REGION Network 1
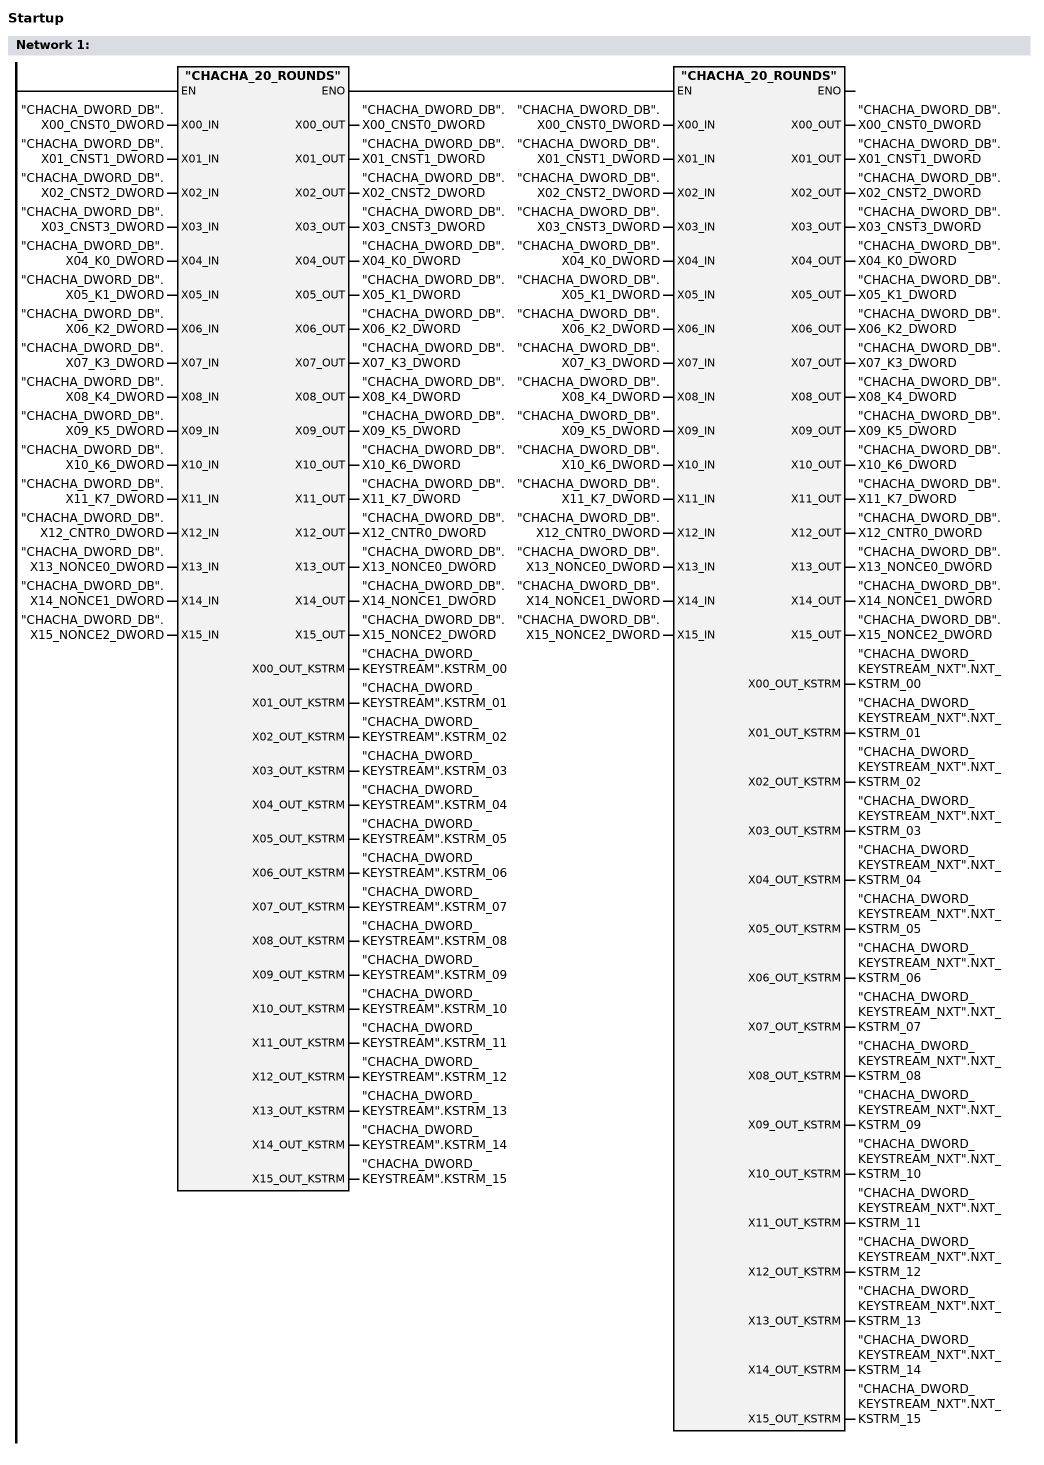
   RUNG wire#powerrail
      "CHACHA_20_ROUNDS"(X00_IN := "CHACHA_DWORD_DB".X00_CNST0_DWORD, X01_IN := "CHACHA_DWORD_DB".X01_CNST1_DWORD, X02_IN := "CHACHA_DWORD_DB".X02_CNST2_DWORD, X03_IN := "CHACHA_DWORD_DB".X03_CNST3_DWORD, X04_IN := "CHACHA_DWORD_DB".X04_K0_DWORD, X05_IN := "CHACHA_DWORD_DB".X05_K1_DWORD, X06_IN := "CHACHA_DWORD_DB".X06_K2_DWORD, X07_IN := "CHACHA_DWORD_DB".X07_K3_DWORD, X08_IN := "CHACHA_DWORD_DB".X08_K4_DWORD, X09_IN := "CHACHA_DWORD_DB".X09_K5_DWORD, X10_IN := "CHACHA_DWORD_DB".X10_K6_DWORD, X11_IN := "CHACHA_DWORD_DB".X11_K7_DWORD, X12_IN := "CHACHA_DWORD_DB".X12_CNTR0_DWORD, X13_IN := "CHACHA_DWORD_DB".X13_NONCE0_DWORD, X14_IN := "CHACHA_DWORD_DB".X14_NONCE1_DWORD, X15_IN := "CHACHA_DWORD_DB".X15_NONCE2_DWORD, X00_OUT => "CHACHA_DWORD_DB".X00_CNST0_DWORD, X01_OUT => "CHACHA_DWORD_DB".X01_CNST1_DWORD, X02_OUT => "CHACHA_DWORD_DB".X02_CNST2_DWORD, X03_OUT => "CHACHA_DWORD_DB".X03_CNST3_DWORD, X04_OUT => "CHACHA_DWORD_DB".X04_K0_DWORD, X05_OUT => "CHACHA_DWORD_DB".X05_K1_DWORD, X06_OUT => "CHACHA_DWORD_DB".X06_K2_DWORD, X07_OUT => "CHACHA_DWORD_DB".X07_K3_DWORD, X08_OUT => "CHACHA_DWORD_DB".X08_K4_DWORD, X09_OUT => "CHACHA_DWORD_DB".X09_K5_DWORD, X10_OUT => "CHACHA_DWORD_DB".X10_K6_DWORD, X11_OUT => "CHACHA_DWORD_DB".X11_K7_DWORD, X12_OUT => "CHACHA_DWORD_DB".X12_CNTR0_DWORD, X13_OUT => "CHACHA_DWORD_DB".X13_NONCE0_DWORD, X14_OUT => "CHACHA_DWORD_DB".X14_NONCE1_DWORD, X15_OUT => "CHACHA_DWORD_DB".X15_NONCE2_DWORD, X00_OUT_KSTRM => "CHACHA_DWORD_KEYSTREAM".KSTRM_00, X01_OUT_KSTRM => "CHACHA_DWORD_KEYSTREAM".KSTRM_01, X02_OUT_KSTRM => "CHACHA_DWORD_KEYSTREAM".KSTRM_02, X03_OUT_KSTRM => "CHACHA_DWORD_KEYSTREAM".KSTRM_03, X04_OUT_KSTRM => "CHACHA_DWORD_KEYSTREAM".KSTRM_04, X05_OUT_KSTRM => "CHACHA_DWORD_KEYSTREAM".KSTRM_05, X06_OUT_KSTRM => "CHACHA_DWORD_KEYSTREAM".KSTRM_06, X07_OUT_KSTRM => "CHACHA_DWORD_KEYSTREAM".KSTRM_07, X08_OUT_KSTRM => "CHACHA_DWORD_KEYSTREAM".KSTRM_08, X09_OUT_KSTRM => "CHACHA_DWORD_KEYSTREAM".KSTRM_09, X10_OUT_KSTRM => "CHACHA_DWORD_KEYSTREAM".KSTRM_10, X11_OUT_KSTRM => "CHACHA_DWORD_KEYSTREAM".KSTRM_11, X12_OUT_KSTRM => "CHACHA_DWORD_KEYSTREAM".KSTRM_12, X13_OUT_KSTRM => "CHACHA_DWORD_KEYSTREAM".KSTRM_13, X14_OUT_KSTRM => "CHACHA_DWORD_KEYSTREAM".KSTRM_14, X15_OUT_KSTRM => "CHACHA_DWORD_KEYSTREAM".KSTRM_15)
      "CHACHA_20_ROUNDS"(X00_IN := "CHACHA_DWORD_DB".X00_CNST0_DWORD, X01_IN := "CHACHA_DWORD_DB".X01_CNST1_DWORD, X02_IN := "CHACHA_DWORD_DB".X02_CNST2_DWORD, X03_IN := "CHACHA_DWORD_DB".X03_CNST3_DWORD, X04_IN := "CHACHA_DWORD_DB".X04_K0_DWORD, X05_IN := "CHACHA_DWORD_DB".X05_K1_DWORD, X06_IN := "CHACHA_DWORD_DB".X06_K2_DWORD, X07_IN := "CHACHA_DWORD_DB".X07_K3_DWORD, X08_IN := "CHACHA_DWORD_DB".X08_K4_DWORD, X09_IN := "CHACHA_DWORD_DB".X09_K5_DWORD, X10_IN := "CHACHA_DWORD_DB".X10_K6_DWORD, X11_IN := "CHACHA_DWORD_DB".X11_K7_DWORD, X12_IN := "CHACHA_DWORD_DB".X12_CNTR0_DWORD, X13_IN := "CHACHA_DWORD_DB".X13_NONCE0_DWORD, X14_IN := "CHACHA_DWORD_DB".X14_NONCE1_DWORD, X15_IN := "CHACHA_DWORD_DB".X15_NONCE2_DWORD, X00_OUT => "CHACHA_DWORD_DB".X00_CNST0_DWORD, X01_OUT => "CHACHA_DWORD_DB".X01_CNST1_DWORD, X02_OUT => "CHACHA_DWORD_DB".X02_CNST2_DWORD, X03_OUT => "CHACHA_DWORD_DB".X03_CNST3_DWORD, X04_OUT => "CHACHA_DWORD_DB".X04_K0_DWORD, X05_OUT => "CHACHA_DWORD_DB".X05_K1_DWORD, X06_OUT => "CHACHA_DWORD_DB".X06_K2_DWORD, X07_OUT => "CHACHA_DWORD_DB".X07_K3_DWORD, X08_OUT => "CHACHA_DWORD_DB".X08_K4_DWORD, X09_OUT => "CHACHA_DWORD_DB".X09_K5_DWORD, X10_OUT => "CHACHA_DWORD_DB".X10_K6_DWORD, X11_OUT => "CHACHA_DWORD_DB".X11_K7_DWORD, X12_OUT => "CHACHA_DWORD_DB".X12_CNTR0_DWORD, X13_OUT => "CHACHA_DWORD_DB".X13_NONCE0_DWORD, X14_OUT => "CHACHA_DWORD_DB".X14_NONCE1_DWORD, X15_OUT => "CHACHA_DWORD_DB".X15_NONCE2_DWORD, X00_OUT_KSTRM => "CHACHA_DWORD_KEYSTREAM_NXT".NXT_KSTRM_00, X01_OUT_KSTRM => "CHACHA_DWORD_KEYSTREAM_NXT".NXT_KSTRM_01, X02_OUT_KSTRM => "CHACHA_DWORD_KEYSTREAM_NXT".NXT_KSTRM_02, X03_OUT_KSTRM => "CHACHA_DWORD_KEYSTREAM_NXT".NXT_KSTRM_03, X04_OUT_KSTRM => "CHACHA_DWORD_KEYSTREAM_NXT".NXT_KSTRM_04, X05_OUT_KSTRM => "CHACHA_DWORD_KEYSTREAM_NXT".NXT_KSTRM_05, X06_OUT_KSTRM => "CHACHA_DWORD_KEYSTREAM_NXT".NXT_KSTRM_06, X07_OUT_KSTRM => "CHACHA_DWORD_KEYSTREAM_NXT".NXT_KSTRM_07, X08_OUT_KSTRM => "CHACHA_DWORD_KEYSTREAM_NXT".NXT_KSTRM_08, X09_OUT_KSTRM => "CHACHA_DWORD_KEYSTREAM_NXT".NXT_KSTRM_09, X10_OUT_KSTRM => "CHACHA_DWORD_KEYSTREAM_NXT".NXT_KSTRM_10, X11_OUT_KSTRM => "CHACHA_DWORD_KEYSTREAM_NXT".NXT_KSTRM_11, X12_OUT_KSTRM => "CHACHA_DWORD_KEYSTREAM_NXT".NXT_KSTRM_12, X13_OUT_KSTRM => "CHACHA_DWORD_KEYSTREAM_NXT".NXT_KSTRM_13, X14_OUT_KSTRM => "CHACHA_DWORD_KEYSTREAM_NXT".NXT_KSTRM_14, X15_OUT_KSTRM => "CHACHA_DWORD_KEYSTREAM_NXT".NXT_KSTRM_15)
   END_RUNG
   // the same network as SCL:
   "CHACHA_20_ROUNDS"(X00_IN := "CHACHA_DWORD_DB".X00_CNST0_DWORD,
                      X01_IN := "CHACHA_DWORD_DB".X01_CNST1_DWORD,
                      X02_IN := "CHACHA_DWORD_DB".X02_CNST2_DWORD,
                      X03_IN := "CHACHA_DWORD_DB".X03_CNST3_DWORD,
                      X04_IN := "CHACHA_DWORD_DB".X04_K0_DWORD,
                      X05_IN := "CHACHA_DWORD_DB".X05_K1_DWORD,
                      X06_IN := "CHACHA_DWORD_DB".X06_K2_DWORD,
                      X07_IN := "CHACHA_DWORD_DB".X07_K3_DWORD,
                      X08_IN := "CHACHA_DWORD_DB".X08_K4_DWORD,
                      X09_IN := "CHACHA_DWORD_DB".X09_K5_DWORD,
                      X10_IN := "CHACHA_DWORD_DB".X10_K6_DWORD,
                      X11_IN := "CHACHA_DWORD_DB".X11_K7_DWORD,
                      X12_IN := "CHACHA_DWORD_DB".X12_CNTR0_DWORD,
                      X13_IN := "CHACHA_DWORD_DB".X13_NONCE0_DWORD,
                      X14_IN := "CHACHA_DWORD_DB".X14_NONCE1_DWORD,
                      X15_IN := "CHACHA_DWORD_DB".X15_NONCE2_DWORD,
                      X00_OUT => "CHACHA_DWORD_DB".X00_CNST0_DWORD,
                      X01_OUT => "CHACHA_DWORD_DB".X01_CNST1_DWORD,
                      X02_OUT => "CHACHA_DWORD_DB".X02_CNST2_DWORD,
                      X03_OUT => "CHACHA_DWORD_DB".X03_CNST3_DWORD,
                      X04_OUT => "CHACHA_DWORD_DB".X04_K0_DWORD,
                      X05_OUT => "CHACHA_DWORD_DB".X05_K1_DWORD,
                      X06_OUT => "CHACHA_DWORD_DB".X06_K2_DWORD,
                      X07_OUT => "CHACHA_DWORD_DB".X07_K3_DWORD,
                      X08_OUT => "CHACHA_DWORD_DB".X08_K4_DWORD,
                      X09_OUT => "CHACHA_DWORD_DB".X09_K5_DWORD,
                      X10_OUT => "CHACHA_DWORD_DB".X10_K6_DWORD,
                      X11_OUT => "CHACHA_DWORD_DB".X11_K7_DWORD,
                      X12_OUT => "CHACHA_DWORD_DB".X12_CNTR0_DWORD,
                      X13_OUT => "CHACHA_DWORD_DB".X13_NONCE0_DWORD,
                      X14_OUT => "CHACHA_DWORD_DB".X14_NONCE1_DWORD,
                      X15_OUT => "CHACHA_DWORD_DB".X15_NONCE2_DWORD,
                      X00_OUT_KSTRM => "CHACHA_DWORD_KEYSTREAM".KSTRM_00,
                      X01_OUT_KSTRM => "CHACHA_DWORD_KEYSTREAM".KSTRM_01,
                      X02_OUT_KSTRM => "CHACHA_DWORD_KEYSTREAM".KSTRM_02,
                      X03_OUT_KSTRM => "CHACHA_DWORD_KEYSTREAM".KSTRM_03,
                      X04_OUT_KSTRM => "CHACHA_DWORD_KEYSTREAM".KSTRM_04,
                      X05_OUT_KSTRM => "CHACHA_DWORD_KEYSTREAM".KSTRM_05,
                      X06_OUT_KSTRM => "CHACHA_DWORD_KEYSTREAM".KSTRM_06,
                      X07_OUT_KSTRM => "CHACHA_DWORD_KEYSTREAM".KSTRM_07,
                      X08_OUT_KSTRM => "CHACHA_DWORD_KEYSTREAM".KSTRM_08,
                      X09_OUT_KSTRM => "CHACHA_DWORD_KEYSTREAM".KSTRM_09,
                      X10_OUT_KSTRM => "CHACHA_DWORD_KEYSTREAM".KSTRM_10,
                      X11_OUT_KSTRM => "CHACHA_DWORD_KEYSTREAM".KSTRM_11,
                      X12_OUT_KSTRM => "CHACHA_DWORD_KEYSTREAM".KSTRM_12,
                      X13_OUT_KSTRM => "CHACHA_DWORD_KEYSTREAM".KSTRM_13,
                      X14_OUT_KSTRM => "CHACHA_DWORD_KEYSTREAM".KSTRM_14,
                      X15_OUT_KSTRM => "CHACHA_DWORD_KEYSTREAM".KSTRM_15,
                      ENO => #_w1);
   IF #_w1 THEN
       "CHACHA_20_ROUNDS"(X00_IN := "CHACHA_DWORD_DB".X00_CNST0_DWORD,
                          X01_IN := "CHACHA_DWORD_DB".X01_CNST1_DWORD,
                          X02_IN := "CHACHA_DWORD_DB".X02_CNST2_DWORD,
                          X03_IN := "CHACHA_DWORD_DB".X03_CNST3_DWORD,
                          X04_IN := "CHACHA_DWORD_DB".X04_K0_DWORD,
                          X05_IN := "CHACHA_DWORD_DB".X05_K1_DWORD,
                          X06_IN := "CHACHA_DWORD_DB".X06_K2_DWORD,
                          X07_IN := "CHACHA_DWORD_DB".X07_K3_DWORD,
                          X08_IN := "CHACHA_DWORD_DB".X08_K4_DWORD,
                          X09_IN := "CHACHA_DWORD_DB".X09_K5_DWORD,
                          X10_IN := "CHACHA_DWORD_DB".X10_K6_DWORD,
                          X11_IN := "CHACHA_DWORD_DB".X11_K7_DWORD,
                          X12_IN := "CHACHA_DWORD_DB".X12_CNTR0_DWORD,
                          X13_IN := "CHACHA_DWORD_DB".X13_NONCE0_DWORD,
                          X14_IN := "CHACHA_DWORD_DB".X14_NONCE1_DWORD,
                          X15_IN := "CHACHA_DWORD_DB".X15_NONCE2_DWORD,
                          X00_OUT => "CHACHA_DWORD_DB".X00_CNST0_DWORD,
                          X01_OUT => "CHACHA_DWORD_DB".X01_CNST1_DWORD,
                          X02_OUT => "CHACHA_DWORD_DB".X02_CNST2_DWORD,
                          X03_OUT => "CHACHA_DWORD_DB".X03_CNST3_DWORD,
                          X04_OUT => "CHACHA_DWORD_DB".X04_K0_DWORD,
                          X05_OUT => "CHACHA_DWORD_DB".X05_K1_DWORD,
                          X06_OUT => "CHACHA_DWORD_DB".X06_K2_DWORD,
                          X07_OUT => "CHACHA_DWORD_DB".X07_K3_DWORD,
                          X08_OUT => "CHACHA_DWORD_DB".X08_K4_DWORD,
                          X09_OUT => "CHACHA_DWORD_DB".X09_K5_DWORD,
                          X10_OUT => "CHACHA_DWORD_DB".X10_K6_DWORD,
                          X11_OUT => "CHACHA_DWORD_DB".X11_K7_DWORD,
                          X12_OUT => "CHACHA_DWORD_DB".X12_CNTR0_DWORD,
                          X13_OUT => "CHACHA_DWORD_DB".X13_NONCE0_DWORD,
                          X14_OUT => "CHACHA_DWORD_DB".X14_NONCE1_DWORD,
                          X15_OUT => "CHACHA_DWORD_DB".X15_NONCE2_DWORD,
                          X00_OUT_KSTRM => "CHACHA_DWORD_KEYSTREAM_NXT".NXT_KSTRM_00,
                          X01_OUT_KSTRM => "CHACHA_DWORD_KEYSTREAM_NXT".NXT_KSTRM_01,
                          X02_OUT_KSTRM => "CHACHA_DWORD_KEYSTREAM_NXT".NXT_KSTRM_02,
                          X03_OUT_KSTRM => "CHACHA_DWORD_KEYSTREAM_NXT".NXT_KSTRM_03,
                          X04_OUT_KSTRM => "CHACHA_DWORD_KEYSTREAM_NXT".NXT_KSTRM_04,
                          X05_OUT_KSTRM => "CHACHA_DWORD_KEYSTREAM_NXT".NXT_KSTRM_05,
                          X06_OUT_KSTRM => "CHACHA_DWORD_KEYSTREAM_NXT".NXT_KSTRM_06,
                          X07_OUT_KSTRM => "CHACHA_DWORD_KEYSTREAM_NXT".NXT_KSTRM_07,
                          X08_OUT_KSTRM => "CHACHA_DWORD_KEYSTREAM_NXT".NXT_KSTRM_08,
                          X09_OUT_KSTRM => "CHACHA_DWORD_KEYSTREAM_NXT".NXT_KSTRM_09,
                          X10_OUT_KSTRM => "CHACHA_DWORD_KEYSTREAM_NXT".NXT_KSTRM_10,
                          X11_OUT_KSTRM => "CHACHA_DWORD_KEYSTREAM_NXT".NXT_KSTRM_11,
                          X12_OUT_KSTRM => "CHACHA_DWORD_KEYSTREAM_NXT".NXT_KSTRM_12,
                          X13_OUT_KSTRM => "CHACHA_DWORD_KEYSTREAM_NXT".NXT_KSTRM_13,
                          X14_OUT_KSTRM => "CHACHA_DWORD_KEYSTREAM_NXT".NXT_KSTRM_14,
                          X15_OUT_KSTRM => "CHACHA_DWORD_KEYSTREAM_NXT".NXT_KSTRM_15);
   END_IF;
END_REGION
END_ORGANIZATION_BLOCK

// ===== PLC "PLC_1"  CPU 1214C AC/DC/Rly =====

VAR_GLOBAL   // PLC tag table "CHACHA"
   "ROUND_001" AT %M41.0 : Bool;
   "CHACHA_001" AT %M41.1 : Bool;
   "ROUND_002" AT %M41.2 : Bool;
   "CHACHA_002" AT %M41.3 : Bool;
   "ROUND_003" AT %M41.4 : Bool;
   "CHACHA_003" AT %M41.5 : Bool;
   "ROUND_004" AT %M41.6 : Bool;
   "CHACHA_004" AT %M41.7 : Bool;
   "ROUND_005" AT %M42.0 : Bool;
   "CHACHA_005" AT %M42.1 : Bool;
   "ROUND_006" AT %M42.2 : Bool;
   "CHACHA_006" AT %M42.3 : Bool;
   "ROUND_007" AT %M42.4 : Bool;
   "CHACHA_007" AT %M42.5 : Bool;
   "ROUND_008" AT %M42.6 : Bool;
   "CHACHA_008" AT %M42.7 : Bool;
   "ROUND_009" AT %M43.0 : Bool;
   "CHACHA_009" AT %M43.1 : Bool;
   "ROUND_010" AT %M43.2 : Bool;
   "CHACHA_010" AT %M43.3 : Bool;
END_VAR

VAR_GLOBAL   // PLC tag table "MUX_KSTRM"
   "KSTRM_NUMBER_DINT" AT %MW33 : UInt;
END_VAR

VAR_GLOBAL   // PLC tag table "TEMP"
   "TEMP_RES" AT %MD64 : DWord;
   "PULSE_TESTE" AT %M120.0 : Bool;
   "PULSE_CHACHA" AT %M120.1 : Bool;
   "PULSE_SEND_START" AT %M120.2 : Bool;
   "PULSE_RCV" AT %M120.3 : Bool;
   "SEND_DATA" AT %M120.4 : Bool;
   "RCV_DATA" AT %M120.5 : Bool;
   "ENABLE_RCV" AT %M120.6 : Bool;
   "ENABLE_CHACHA" AT %M120.7 : Bool;
   "DISABLE_WHILE_CHACHA" AT %M121.0 : Bool;
   "DISABLE_ADD" AT %M121.1 : Bool;
   "SEND_ERROR" AT %M121.2 : Bool;
   "SEND_DONE" AT %M121.3 : Bool;
   "DISABLE_TESTE" AT %M5.0 : Bool;
   "RCV_ERROR" AT %M5.1 : Bool;
   "SEND_STATUS" AT %MW10 : UInt;
   "PULSE_SEND_DONE" AT %M121.4 : Bool;
   "RCV_STATUS" AT %MW12 : UInt;
END_VAR

VAR_GLOBAL   // PLC tag table "QR_FRAC"
   "P_001" AT %M40.0 : Bool;
   "P_002" AT %M40.1 : Bool;
   "P_003" AT %M40.2 : Bool;
   "P_004" AT %M40.3 : Bool;
   "P_005" AT %M40.4 : Bool;
   "P_006" AT %M40.5 : Bool;
   "P_007" AT %M40.6 : Bool;
   "P_008" AT %M40.7 : Bool;
   "P_TRIGGER_001" AT %M20.0 : Bool;
   "P_TRIGGER_002" AT %M20.1 : Bool;
   "P_TRIGGER_003" AT %M20.2 : Bool;
   "P_TRIGGER_004" AT %M20.3 : Bool;
   "P_TRIGGER_005" AT %M20.4 : Bool;
   "P_TRIGGER_006" AT %M20.5 : Bool;
   "P_TRIGGER_007" AT %M20.6 : Bool;
   "P_TRIGGER_008" AT %M20.7 : Bool;
END_VAR

VAR_GLOBAL   // PLC tag table "QR"
   "QR_P001" AT %M21.0 : Bool;
   "QR_P002" AT %M21.1 : Bool;
   "QR_P003" AT %M21.2 : Bool;
   "QR_P004" AT %M21.3 : Bool;
   "QR_TRIGGER001" AT %M21.4 : Bool;
   "QR_TRIGGER002" AT %M21.5 : Bool;
   "QR_TRIGGER003" AT %M21.6 : Bool;
   "QR_TRIGGER004" AT %M21.7 : Bool;
END_VAR

VAR_GLOBAL   // PLC tag table "QR_COL"
   "QRCOL_P001" AT %M22.0 : Bool;
   "QRCOL_P002" AT %M22.1 : Bool;
   "QRCOL_P003" AT %M22.2 : Bool;
   "QRCOL_P004" AT %M22.3 : Bool;
   "QRCOL_TRG001" AT %M22.4 : Bool;
   "QRCOL_TRG002" AT %M22.5 : Bool;
   "QRCOL_TRG003" AT %M22.6 : Bool;
   "QRCOL_TRG004" AT %M22.7 : Bool;
END_VAR

VAR_GLOBAL   // PLC tag table "QR_DIAG"
   "QRDIAG_P001" AT %M23.0 : Bool;
   "QRDIAG_P002" AT %M23.1 : Bool;
   "QRDIAG_P003" AT %M23.2 : Bool;
   "QRDIAG_P004" AT %M23.3 : Bool;
   "QRDIAG_TRG001" AT %M23.4 : Bool;
   "QRDIAG_TRG002" AT %M23.5 : Bool;
   "QRDIAG_TRG003" AT %M23.6 : Bool;
   "QRDIAG_TRG004" AT %M23.7 : Bool;
END_VAR

VAR_GLOBAL   // PLC tag table "CHACHA_1R"
   "1R_P001" AT %M24.0 : Bool;
   "1R_P002" AT %M24.1 : Bool;
   "1R_P003" AT %M24.2 : Bool;
   "1R_TRG001" AT %M24.3 : Bool;
   "1R_TRG002" AT %M24.4 : Bool;
   "1R_TRG003" AT %M24.5 : Bool;
END_VAR

VAR_GLOBAL   // PLC tag table "IO_BT"
   "BT_TESTE" AT %I0.0 : Bool;
   "BT_ENABLE_SEND" AT %I0.1 : Bool;
   "BT_ENABLE_RCV" AT %I0.2 : Bool;
   "BT_DATA_SEND" AT %I0.3 : Bool;
   "BT_DATA_RCV" AT %I0.4 : Bool;
   "BT_PLAIN_0" AT %I1.0 : Bool;
   "BT_PLAIN_1" AT %I1.1 : Bool;
   "BT_PLAIN_2" AT %I1.2 : Bool;
   "BT_PLAIN_3" AT %I1.3 : Bool;
   "BT_PLAIN_4" AT %I1.4 : Bool;
   "BT_PLAIN_5" AT %I1.5 : Bool;
END_VAR

DATA_BLOCK "CHACHA_DWORD_KEYSTREAM"   // DB1
{ S7_Optimized_Access := 'TRUE' }
VERSION : 0.1
   VAR
      KSTRM_00 : DWord;
      KSTRM_01 : DWord;
      KSTRM_02 : DWord;
      KSTRM_03 : DWord;
      KSTRM_04 : DWord;
      KSTRM_05 : DWord;
      KSTRM_06 : DWord;
      KSTRM_07 : DWord;
      KSTRM_08 : DWord;
      KSTRM_09 : DWord;
      KSTRM_10 : DWord;
      KSTRM_11 : DWord;
      KSTRM_12 : DWord;
      KSTRM_13 : DWord;
      KSTRM_14 : DWord;
      KSTRM_15 : DWord;
   END_VAR
BEGIN
END_DATA_BLOCK

DATA_BLOCK "CHACHA_DWORD_DB"   // DB2
{ S7_Optimized_Access := 'TRUE' }
VERSION : 0.1
   VAR
      X00_CNST0_DWORD : DWord := 16#6170_7865;
      X01_CNST1_DWORD : DWord := 16#3320_646E;
      X02_CNST2_DWORD : DWord := 16#7962_2D32;
      X03_CNST3_DWORD : DWord := 16#6B20_6574;
      X04_K0_DWORD : DWord := 16#0101_1100;
      X05_K1_DWORD : DWord := 16#0010_0110;
      X06_K2_DWORD : DWord := 16#1110_0000;
      X07_K3_DWORD : DWord := 16#0001_1110;
      X08_K4_DWORD : DWord := 16#0110_0010;
      X09_K5_DWORD : DWord := 16#1010_0101;
      X10_K6_DWORD : DWord := 16#0001_1000;
      X11_K7_DWORD : DWord := 16#0110_0110;
      X12_CNTR0_DWORD : DWord := 16#0000_0000;
      X13_NONCE0_DWORD : DWord := 16#0011_1100;
      X14_NONCE1_DWORD : DWord := 16#0101_1010;
      X15_NONCE2_DWORD : DWord := 16#1111_1111;
   END_VAR
BEGIN
END_DATA_BLOCK

DATA_BLOCK "CHACHA_DWORD_PLAINTXT"   // DB3
{ S7_Optimized_Access := 'TRUE' }
VERSION : 0.1
   VAR
      X00_PLAINTXT_RCV : DWord;
      X00_PLAINTXT_SEND : DWord;
   END_VAR
BEGIN
END_DATA_BLOCK

DATA_BLOCK "CHACHA_DWORD_CIPHERTXT"   // DB4
{ S7_Optimized_Access := 'FALSE' }
VERSION : 0.1
   VAR
      X00_CIPHERTXT : DWord;
   END_VAR
BEGIN
END_DATA_BLOCK

DATA_BLOCK "RUNTIME"   // DB7
{ S7_Optimized_Access := 'TRUE' }
VERSION : 0.1
   VAR
      RTIME_00 : LReal;
      RTIME_RES_00 : LReal;
   END_VAR
BEGIN
END_DATA_BLOCK

DATA_BLOCK "MUX_KSTRM"   // DB10
{ S7_Optimized_Access := 'TRUE' }
VERSION : 0.1
   VAR
      KSTRM_NUMBER_DINT : DInt := 0;
      KSTRM_USE : DWord;
   END_VAR
BEGIN
END_DATA_BLOCK

DATA_BLOCK "CHACHA_DWORD_KEYSTREAM_NXT"   // DB11
{ S7_Optimized_Access := 'TRUE' }
VERSION : 0.1
   VAR
      NXT_KSTRM_00 : DWord;
      NXT_KSTRM_01 : DWord;
      NXT_KSTRM_02 : DWord;
      NXT_KSTRM_03 : DWord;
      NXT_KSTRM_04 : DWord;
      NXT_KSTRM_05 : DWord;
      NXT_KSTRM_06 : DWord;
      NXT_KSTRM_07 : DWord;
      NXT_KSTRM_08 : DWord;
      NXT_KSTRM_09 : DWord;
      NXT_KSTRM_10 : DWord;
      NXT_KSTRM_11 : DWord;
      NXT_KSTRM_12 : DWord;
      NXT_KSTRM_13 : DWord;
      NXT_KSTRM_14 : DWord;
      NXT_KSTRM_15 : DWord;
   END_VAR
BEGIN
END_DATA_BLOCK

DATA_BLOCK "RETENTIVE_TAGS"   // DB12
{ S7_Optimized_Access := 'TRUE' }
VERSION : 0.1
   VAR
      ENABLE_CHACHA : Bool;
      "DISABLE WHILE CHACHA" : Bool;
      BUSY_SEND : Bool;
   END_VAR
BEGIN
END_DATA_BLOCK

// folder: System blocks/Program resources

DATA_BLOCK "PLC_2_Send_DB"   // DB8
{ S7_Optimized_Access := 'TRUE' }
AUTHOR : SIMATIC
FAMILY : MC7Plus
NAME : TCON_Prm
VERSION : 1.0
// stored: InstanceOfName TCON_Param
"TCON_Param"
BEGIN
   ID := 1;
   REM_TSAP_ID[1] := B#16#07;
   REM_TSAP_ID[2] := B#16#D0;
   REM_STADDR[1] := 192;
   REM_STADDR[2] := 168;
   REM_STADDR[4] := 2;
END_DATA_BLOCK

DATA_BLOCK "PLC_2_Receive_DB"   // DB9
{ S7_Optimized_Access := 'TRUE' }
AUTHOR : SIMATIC
FAMILY : MC7Plus
NAME : TCON_Prm
VERSION : 1.0
// stored: InstanceOfName TCON_Param
"TCON_Param"
BEGIN
   ID := 2;
   REM_TSAP_ID_LEN := 0;
   LOCAL_TSAP_ID[1] := B#16#07;
   LOCAL_TSAP_ID[2] := B#16#D0;
   LOCAL_TSAP_ID_LEN := 2;
   ACTIVE_EST := false;
   REM_STADDR[1] := 192;
   REM_STADDR[2] := 168;
   REM_STADDR[4] := 2;
END_DATA_BLOCK

// folder: (top level)

FUNCTION "QR" : Void   // FC1, LAD
{ S7_Optimized_Access := 'TRUE' }
VERSION : 0.1
   VAR_INPUT
      IN_ZA : DWord;
      IN_ZB : DWord;
      IN_ZC : DWord;
      IN_ZD : DWord;
   END_VAR
   VAR_OUTPUT
      OUT_ZA : DWord;
      OUT_ZB : DWord;
      OUT_ZC : DWord;
      OUT_ZD : DWord;
   END_VAR
   VAR_TEMP
      TEMP_ZA : DWord;
      TEMP_ZB : DWord;
      TEMP_ZC : DWord;
      TEMP_ZD : DWord;
   END_VAR
   VAR_TEMP   // added for the SCL form of the ladder/FBD networks
      _w1 : Bool;
   END_VAR
BEGIN

REGION Network 1
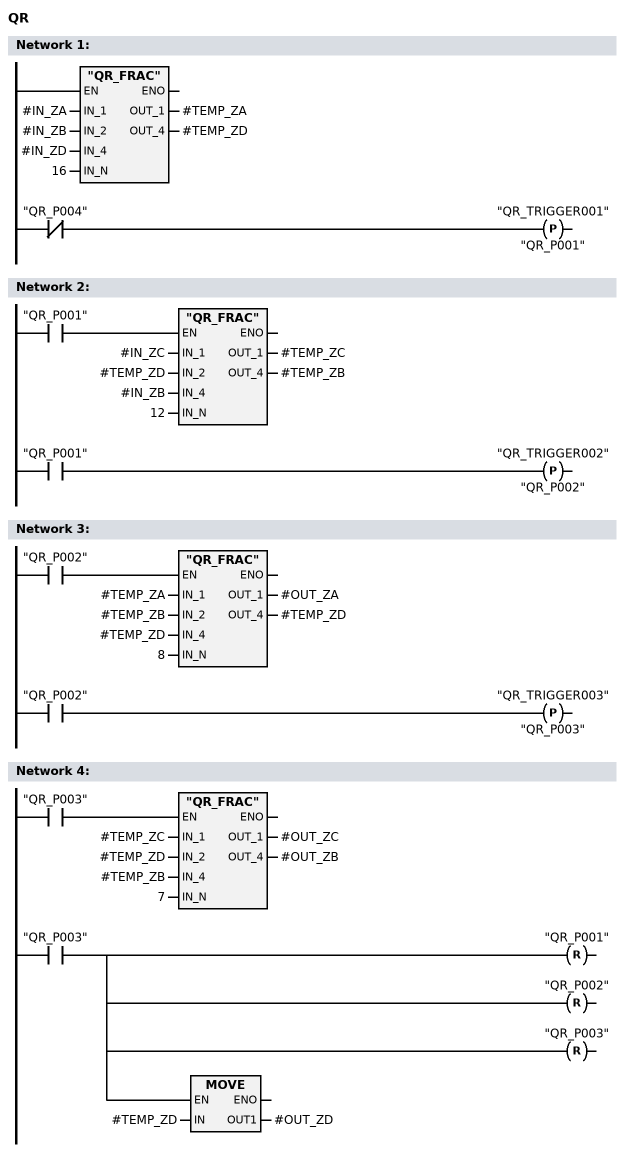
   "QR_FRAC"(IN_1 := #IN_ZA, IN_2 := #IN_ZB, IN_4 := #IN_ZD, IN_N := 16, OUT_1 => #TEMP_ZA, OUT_4 => #TEMP_ZD);
   "QR_TRIGGER001" := NOT "QR_P004" AND NOT "QR_P001";   // rising edge
   "QR_P001" := NOT "QR_P004";
END_REGION

REGION Network 2
   IF "QR_P001" THEN
       "QR_FRAC"(IN_1 := #IN_ZC, IN_2 := #TEMP_ZD, IN_4 := #IN_ZB, IN_N := 12, OUT_1 => #TEMP_ZC, OUT_4 => #TEMP_ZB);
   END_IF;
   "QR_TRIGGER002" := "QR_P001" AND NOT "QR_P002";   // rising edge
   "QR_P002" := "QR_P001";
END_REGION

REGION Network 3
   IF "QR_P002" THEN
       "QR_FRAC"(IN_1 := #TEMP_ZA,
                 IN_2 := #TEMP_ZB,
                 IN_4 := #TEMP_ZD,
                 IN_N := 8,
                 OUT_1 => #OUT_ZA,
                 OUT_4 => #TEMP_ZD);
   END_IF;
   "QR_TRIGGER003" := "QR_P002" AND NOT "QR_P003";   // rising edge
   "QR_P003" := "QR_P002";
END_REGION

REGION Network 4
   RUNG wire#powerrail
      Contact( "QR_P003" )
      "QR_FRAC"(IN_1 := #TEMP_ZC, IN_2 := #TEMP_ZD, IN_4 := #TEMP_ZB, IN_N := 7, OUT_1 => #OUT_ZC, OUT_4 => #OUT_ZB)
   END_RUNG
   RUNG wire#powerrail
      Contact( "QR_P003" )
      wire#w1
      R_Coil( "QR_P001" )
   END_RUNG
   RUNG wire#w1
      R_Coil( "QR_P002" )
   END_RUNG
   RUNG wire#w1
      R_Coil( "QR_P003" )
   END_RUNG
   RUNG wire#w1
      { S7_GenerateENO := "TRUE" } Move(in := #TEMP_ZD, out1 => #OUT_ZD)
   END_RUNG
   // the same network as SCL:
   IF "QR_P003" THEN
       "QR_FRAC"(IN_1 := #TEMP_ZC,
                 IN_2 := #TEMP_ZD,
                 IN_4 := #TEMP_ZB,
                 IN_N := 7,
                 OUT_1 => #OUT_ZC,
                 OUT_4 => #OUT_ZB);
   END_IF;
   IF "QR_P003" THEN
       "QR_P001" := FALSE;
       "QR_P002" := FALSE;
   END_IF;
   #_w1 := "QR_P003";
   IF #_w1 THEN
       "QR_P003" := FALSE;
       #OUT_ZD := #TEMP_ZD;
   END_IF;
END_REGION
END_FUNCTION

FUNCTION "QR_FRAC" : Void   // FC2, LAD
{ S7_Optimized_Access := 'TRUE' }
VERSION : 0.1
   VAR_INPUT
      IN_1 : DWord;
      IN_2 : DWord;
      IN_4 : DWord;
      IN_N : UInt;
   END_VAR
   VAR_OUTPUT
      OUT_1 : DWord;
      OUT_4 : DWord;
   END_VAR
   VAR_TEMP
      TEMP_1 : DWord;
      TEMP_4 : DWord;
      TEMP_UDINT_1 : UDInt;
      TEMP_UDINT_2 : UDInt;
   END_VAR
BEGIN

REGION Network 1
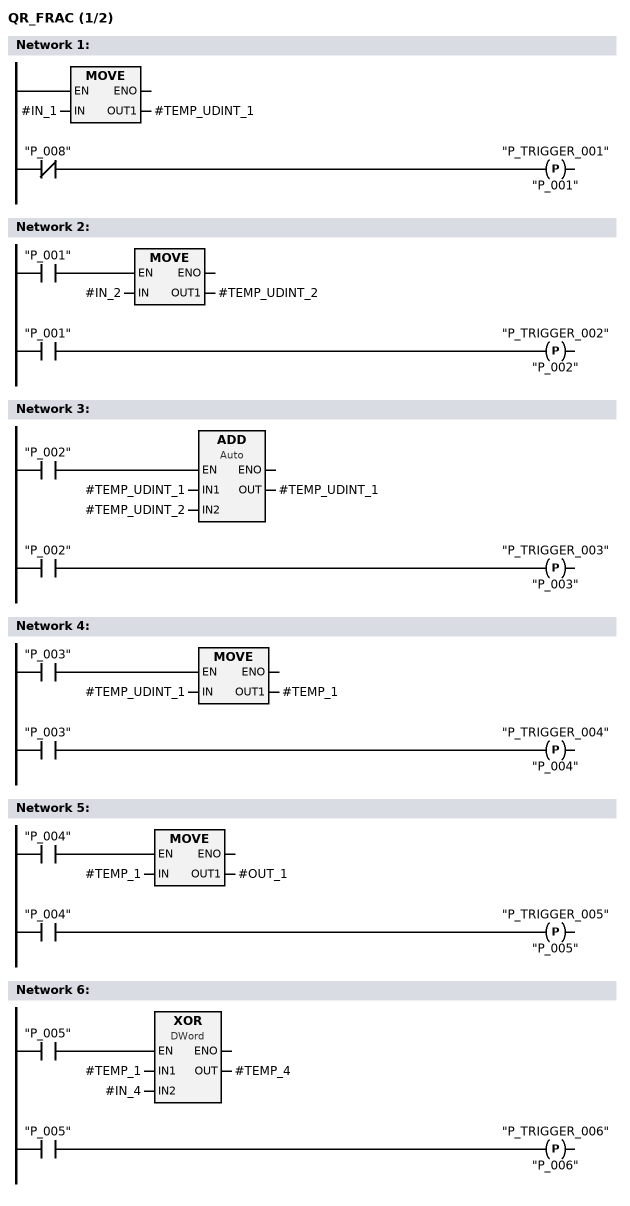
   #TEMP_UDINT_1 := #IN_1;
   "P_TRIGGER_001" := NOT "P_008" AND NOT "P_001";   // rising edge
   "P_001" := NOT "P_008";
END_REGION

REGION Network 2
   IF "P_001" THEN #TEMP_UDINT_2 := #IN_2; END_IF;
   "P_TRIGGER_002" := "P_001" AND NOT "P_002";   // rising edge
   "P_002" := "P_001";
END_REGION

REGION Network 3
   IF "P_002" THEN #TEMP_UDINT_1 := #TEMP_UDINT_1 + #TEMP_UDINT_2; END_IF;
   "P_TRIGGER_003" := "P_002" AND NOT "P_003";   // rising edge
   "P_003" := "P_002";
END_REGION

REGION Network 4
   IF "P_003" THEN #TEMP_1 := #TEMP_UDINT_1; END_IF;
   "P_TRIGGER_004" := "P_003" AND NOT "P_004";   // rising edge
   "P_004" := "P_003";
END_REGION

REGION Network 5
   IF "P_004" THEN #OUT_1 := #TEMP_1; END_IF;
   "P_TRIGGER_005" := "P_004" AND NOT "P_005";   // rising edge
   "P_005" := "P_004";
END_REGION

REGION Network 6
   IF "P_005" THEN #TEMP_4 := #TEMP_1 XOR #IN_4; END_IF;
   "P_TRIGGER_006" := "P_005" AND NOT "P_006";   // rising edge
   "P_006" := "P_005";
END_REGION

REGION Network 7
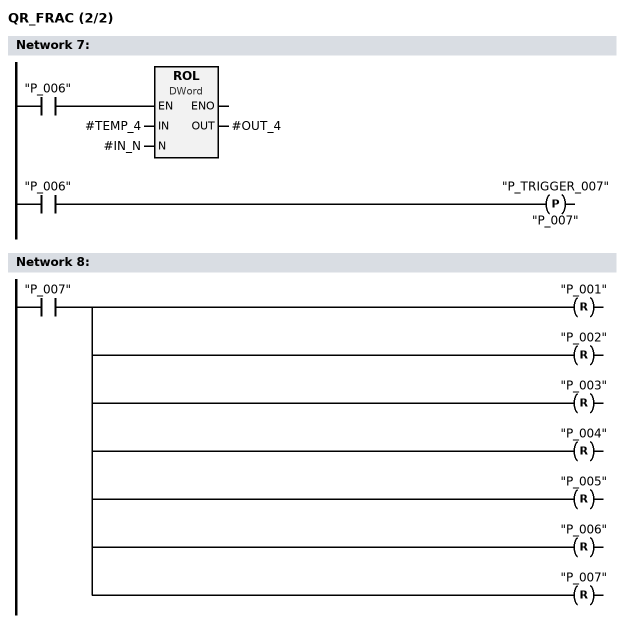
   IF "P_006" THEN #OUT_4 := ROL(IN := #TEMP_4, N := #IN_N); END_IF;
   "P_TRIGGER_007" := "P_006" AND NOT "P_007";   // rising edge
   "P_007" := "P_006";
END_REGION

REGION Network 8
   RUNG wire#powerrail
      Contact( "P_007" )
      wire#w1
      R_Coil( "P_001" )
   END_RUNG
   RUNG wire#w1
      R_Coil( "P_002" )
   END_RUNG
   RUNG wire#w1
      R_Coil( "P_003" )
   END_RUNG
   RUNG wire#w1
      R_Coil( "P_004" )
   END_RUNG
   RUNG wire#w1
      R_Coil( "P_005" )
   END_RUNG
   RUNG wire#w1
      R_Coil( "P_006" )
   END_RUNG
   RUNG wire#w1
      R_Coil( "P_007" )
   END_RUNG
   // the same network as SCL:
   IF "P_007" THEN
       "P_001" := FALSE;
       "P_002" := FALSE;
       "P_003" := FALSE;
       "P_004" := FALSE;
       "P_005" := FALSE;
       "P_006" := FALSE;
       "P_007" := FALSE;
   END_IF;
END_REGION
END_FUNCTION

FUNCTION "QR_COL" : Void   // FC3, LAD
{ S7_Optimized_Access := 'TRUE' }
VERSION : 0.1
   VAR_INPUT
      X00_IN_COL : DWord;
      X01_IN_COL : DWord;
      X02_IN_COL : DWord;
      X03_IN_COL : DWord;
      X04_IN_COL : DWord;
      X05_IN_COL : DWord;
      X06_IN_COL : DWord;
      X07_IN_COL : DWord;
      X08_IN_COL : DWord;
      X09_IN_COL : DWord;
      X10_IN_COL : DWord;
      X11_IN_COL : DWord;
      X12_IN_COL : DWord;
      X13_IN_COL : DWord;
      X14_IN_COL : DWord;
      X15_IN_COL : DWord;
   END_VAR
   VAR_OUTPUT
      X00_OUT_COL : DWord;
      X01_OUT_COL : DWord;
      X02_OUT_COL : DWord;
      X03_OUT_COL : DWord;
      X04_OUT_COL : DWord;
      X05_OUT_COL : DWord;
      X06_OUT_COL : DWord;
      X07_OUT_COL : DWord;
      X08_OUT_COL : DWord;
      X09_OUT_COL : DWord;
      X10_OUT_COL : DWord;
      X11_OUT_COL : DWord;
      X12_OUT_COL : DWord;
      X13_OUT_COL : DWord;
      X14_OUT_COL : DWord;
      X15_OUT_COL : DWord;
   END_VAR
BEGIN

REGION Network 1
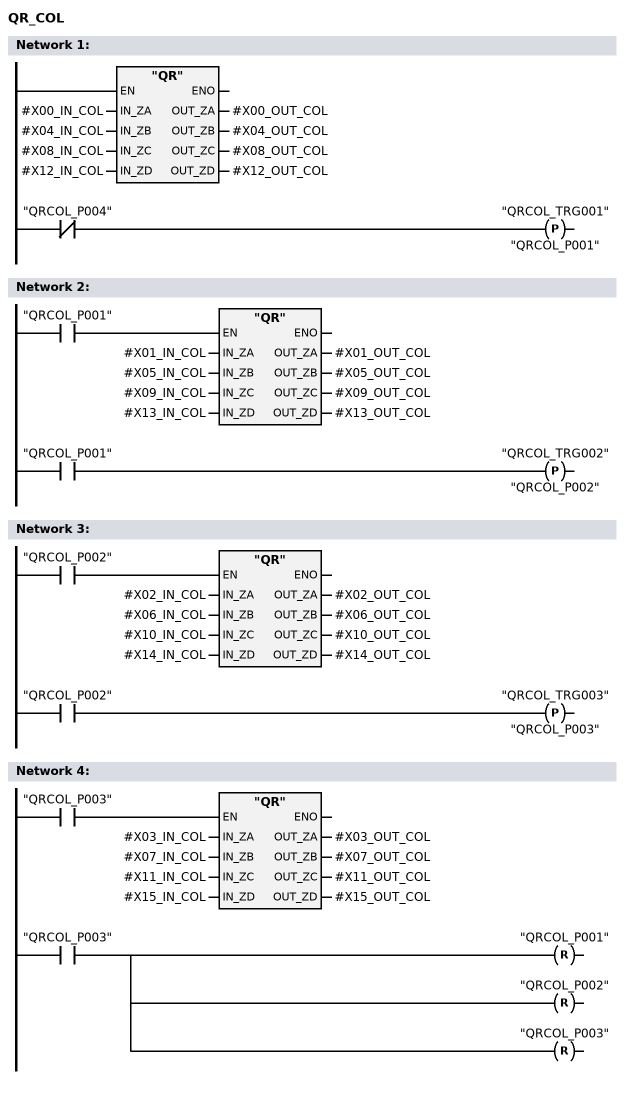
   "QR"(IN_ZA := #X00_IN_COL,
        IN_ZB := #X04_IN_COL,
        IN_ZC := #X08_IN_COL,
        IN_ZD := #X12_IN_COL,
        OUT_ZA => #X00_OUT_COL,
        OUT_ZB => #X04_OUT_COL,
        OUT_ZC => #X08_OUT_COL,
        OUT_ZD => #X12_OUT_COL);
   "QRCOL_TRG001" := NOT "QRCOL_P004" AND NOT "QRCOL_P001";   // rising edge
   "QRCOL_P001" := NOT "QRCOL_P004";
END_REGION

REGION Network 2
   IF "QRCOL_P001" THEN
       "QR"(IN_ZA := #X01_IN_COL,
            IN_ZB := #X05_IN_COL,
            IN_ZC := #X09_IN_COL,
            IN_ZD := #X13_IN_COL,
            OUT_ZA => #X01_OUT_COL,
            OUT_ZB => #X05_OUT_COL,
            OUT_ZC => #X09_OUT_COL,
            OUT_ZD => #X13_OUT_COL);
   END_IF;
   "QRCOL_TRG002" := "QRCOL_P001" AND NOT "QRCOL_P002";   // rising edge
   "QRCOL_P002" := "QRCOL_P001";
END_REGION

REGION Network 3
   IF "QRCOL_P002" THEN
       "QR"(IN_ZA := #X02_IN_COL,
            IN_ZB := #X06_IN_COL,
            IN_ZC := #X10_IN_COL,
            IN_ZD := #X14_IN_COL,
            OUT_ZA => #X02_OUT_COL,
            OUT_ZB => #X06_OUT_COL,
            OUT_ZC => #X10_OUT_COL,
            OUT_ZD => #X14_OUT_COL);
   END_IF;
   "QRCOL_TRG003" := "QRCOL_P002" AND NOT "QRCOL_P003";   // rising edge
   "QRCOL_P003" := "QRCOL_P002";
END_REGION

REGION Network 4
   RUNG wire#powerrail
      Contact( "QRCOL_P003" )
      "QR"(IN_ZA := #X03_IN_COL, IN_ZB := #X07_IN_COL, IN_ZC := #X11_IN_COL, IN_ZD := #X15_IN_COL, OUT_ZA => #X03_OUT_COL, OUT_ZB => #X07_OUT_COL, OUT_ZC => #X11_OUT_COL, OUT_ZD => #X15_OUT_COL)
   END_RUNG
   RUNG wire#powerrail
      Contact( "QRCOL_P003" )
      wire#w1
      R_Coil( "QRCOL_P001" )
   END_RUNG
   RUNG wire#w1
      R_Coil( "QRCOL_P002" )
   END_RUNG
   RUNG wire#w1
      R_Coil( "QRCOL_P003" )
   END_RUNG
   // the same network as SCL:
   IF "QRCOL_P003" THEN
       "QR"(IN_ZA := #X03_IN_COL,
            IN_ZB := #X07_IN_COL,
            IN_ZC := #X11_IN_COL,
            IN_ZD := #X15_IN_COL,
            OUT_ZA => #X03_OUT_COL,
            OUT_ZB => #X07_OUT_COL,
            OUT_ZC => #X11_OUT_COL,
            OUT_ZD => #X15_OUT_COL);
   END_IF;
   IF "QRCOL_P003" THEN
       "QRCOL_P001" := FALSE;
       "QRCOL_P002" := FALSE;
       "QRCOL_P003" := FALSE;
   END_IF;
END_REGION
END_FUNCTION

FUNCTION "QR_DIAG" : Void   // FC4, LAD
{ S7_Optimized_Access := 'TRUE' }
VERSION : 0.1
   VAR_INPUT
      X00_IN_DIAG : DWord;
      X01_IN_DIAG : DWord;
      X02_IN_DIAG : DWord;
      X03_IN_DIAG : DWord;
      X04_IN_DIAG : DWord;
      X05_IN_DIAG : DWord;
      X06_IN_DIAG : DWord;
      X07_IN_DIAG : DWord;
      X08_IN_DIAG : DWord;
      X09_IN_DIAG : DWord;
      X10_IN_DIAG : DWord;
      X11_IN_DIAG : DWord;
      X12_IN_DIAG : DWord;
      X13_IN_DIAG : DWord;
      X14_IN_DIAG : DWord;
      X15_IN_DIAG : DWord;
   END_VAR
   VAR_OUTPUT
      X00_OUT_DIAG : DWord;
      X01_OUT_DIAG : DWord;
      X02_OUT_DIAG : DWord;
      X03_OUT_DIAG : DWord;
      X04_OUT_DIAG : DWord;
      X05_OUT_DIAG : DWord;
      X06_OUT_DIAG : DWord;
      X07_OUT_DIAG : DWord;
      X08_OUT_DIAG : DWord;
      X09_OUT_DIAG : DWord;
      X10_OUT_DIAG : DWord;
      X11_OUT_DIAG : DWord;
      X12_OUT_DIAG : DWord;
      X13_OUT_DIAG : DWord;
      X14_OUT_DIAG : DWord;
      X15_OUT_DIAG : DWord;
   END_VAR
BEGIN

REGION Network 1
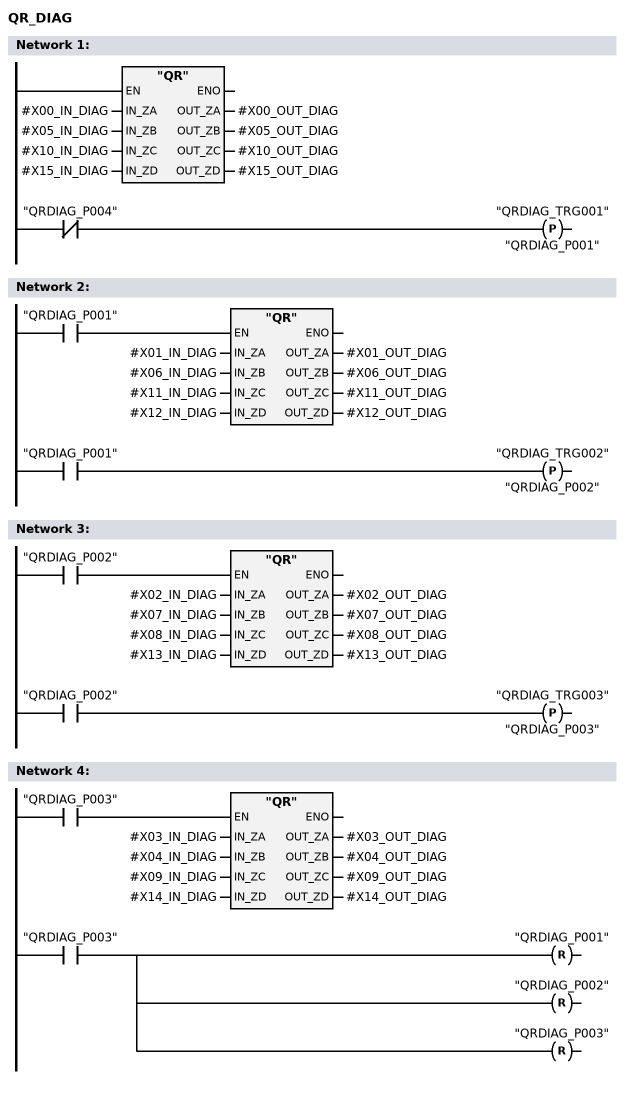
   "QR"(IN_ZA := #X00_IN_DIAG,
        IN_ZB := #X05_IN_DIAG,
        IN_ZC := #X10_IN_DIAG,
        IN_ZD := #X15_IN_DIAG,
        OUT_ZA => #X00_OUT_DIAG,
        OUT_ZB => #X05_OUT_DIAG,
        OUT_ZC => #X10_OUT_DIAG,
        OUT_ZD => #X15_OUT_DIAG);
   "QRDIAG_TRG001" := NOT "QRDIAG_P004" AND NOT "QRDIAG_P001";   // rising edge
   "QRDIAG_P001" := NOT "QRDIAG_P004";
END_REGION

REGION Network 2
   IF "QRDIAG_P001" THEN
       "QR"(IN_ZA := #X01_IN_DIAG,
            IN_ZB := #X06_IN_DIAG,
            IN_ZC := #X11_IN_DIAG,
            IN_ZD := #X12_IN_DIAG,
            OUT_ZA => #X01_OUT_DIAG,
            OUT_ZB => #X06_OUT_DIAG,
            OUT_ZC => #X11_OUT_DIAG,
            OUT_ZD => #X12_OUT_DIAG);
   END_IF;
   "QRDIAG_TRG002" := "QRDIAG_P001" AND NOT "QRDIAG_P002";   // rising edge
   "QRDIAG_P002" := "QRDIAG_P001";
END_REGION

REGION Network 3
   IF "QRDIAG_P002" THEN
       "QR"(IN_ZA := #X02_IN_DIAG,
            IN_ZB := #X07_IN_DIAG,
            IN_ZC := #X08_IN_DIAG,
            IN_ZD := #X13_IN_DIAG,
            OUT_ZA => #X02_OUT_DIAG,
            OUT_ZB => #X07_OUT_DIAG,
            OUT_ZC => #X08_OUT_DIAG,
            OUT_ZD => #X13_OUT_DIAG);
   END_IF;
   "QRDIAG_TRG003" := "QRDIAG_P002" AND NOT "QRDIAG_P003";   // rising edge
   "QRDIAG_P003" := "QRDIAG_P002";
END_REGION

REGION Network 4
   RUNG wire#powerrail
      Contact( "QRDIAG_P003" )
      "QR"(IN_ZA := #X03_IN_DIAG, IN_ZB := #X04_IN_DIAG, IN_ZC := #X09_IN_DIAG, IN_ZD := #X14_IN_DIAG, OUT_ZA => #X03_OUT_DIAG, OUT_ZB => #X04_OUT_DIAG, OUT_ZC => #X09_OUT_DIAG, OUT_ZD => #X14_OUT_DIAG)
   END_RUNG
   RUNG wire#powerrail
      Contact( "QRDIAG_P003" )
      wire#w1
      R_Coil( "QRDIAG_P001" )
   END_RUNG
   RUNG wire#w1
      R_Coil( "QRDIAG_P002" )
   END_RUNG
   RUNG wire#w1
      R_Coil( "QRDIAG_P003" )
   END_RUNG
   // the same network as SCL:
   IF "QRDIAG_P003" THEN
       "QR"(IN_ZA := #X03_IN_DIAG,
            IN_ZB := #X04_IN_DIAG,
            IN_ZC := #X09_IN_DIAG,
            IN_ZD := #X14_IN_DIAG,
            OUT_ZA => #X03_OUT_DIAG,
            OUT_ZB => #X04_OUT_DIAG,
            OUT_ZC => #X09_OUT_DIAG,
            OUT_ZD => #X14_OUT_DIAG);
   END_IF;
   IF "QRDIAG_P003" THEN
       "QRDIAG_P001" := FALSE;
       "QRDIAG_P002" := FALSE;
       "QRDIAG_P003" := FALSE;
   END_IF;
END_REGION
END_FUNCTION

FUNCTION "CHACHA_20_ROUNDS" : Void   // FC5, LAD
{ S7_Optimized_Access := 'TRUE' }
VERSION : 0.1
   VAR_INPUT
      X00_IN : DWord;
      X01_IN : DWord;
      X02_IN : DWord;
      X03_IN : DWord;
      X04_IN : DWord;
      X05_IN : DWord;
      X06_IN : DWord;
      X07_IN : DWord;
      X08_IN : DWord;
      X09_IN : DWord;
      X10_IN : DWord;
      X11_IN : DWord;
      X12_IN : DWord;
      X13_IN : DWord;
      X14_IN : DWord;
      X15_IN : DWord;
   END_VAR
   VAR_OUTPUT
      X00_OUT : DWord;
      X01_OUT : DWord;
      X02_OUT : DWord;
      X03_OUT : DWord;
      X04_OUT : DWord;
      X05_OUT : DWord;
      X06_OUT : DWord;
      X07_OUT : DWord;
      X08_OUT : DWord;
      X09_OUT : DWord;
      X10_OUT : DWord;
      X11_OUT : DWord;
      X12_OUT : DWord;
      X13_OUT : DWord;
      X14_OUT : DWord;
      X15_OUT : DWord;
      X00_OUT_KSTRM : DWord;
      X01_OUT_KSTRM : DWord;
      X02_OUT_KSTRM : DWord;
      X03_OUT_KSTRM : DWord;
      X04_OUT_KSTRM : DWord;
      X05_OUT_KSTRM : DWord;
      X06_OUT_KSTRM : DWord;
      X07_OUT_KSTRM : DWord;
      X08_OUT_KSTRM : DWord;
      X09_OUT_KSTRM : DWord;
      X10_OUT_KSTRM : DWord;
      X11_OUT_KSTRM : DWord;
      X12_OUT_KSTRM : DWord;
      X13_OUT_KSTRM : DWord;
      X14_OUT_KSTRM : DWord;
      X15_OUT_KSTRM : DWord;
   END_VAR
   VAR_TEMP
      TEMP_X00 : DWord;
      TEMP_X01 : DWord;
      TEMP_X02 : DWord;
      TEMP_X03 : DWord;
      TEMP_X04 : DWord;
      TEMP_X05 : DWord;
      TEMP_X06 : DWord;
      TEMP_X07 : DWord;
      TEMP_X08 : DWord;
      TEMP_X09 : DWord;
      TEMP_X10 : DWord;
      TEMP_X11 : DWord;
      TEMP_X12 : DWord;
      TEMP_X13 : DWord;
      TEMP_X14 : DWord;
      TEMP_X15 : DWord;
      TEMP_CNST_INT : UDInt;
      TEMP_CNST_DWORD : DWord;
   END_VAR
   VAR_TEMP   // added for the SCL form of the ladder/FBD networks
      _w1 : Bool;
      _w2 : Bool;
   END_VAR
BEGIN

REGION Network 1
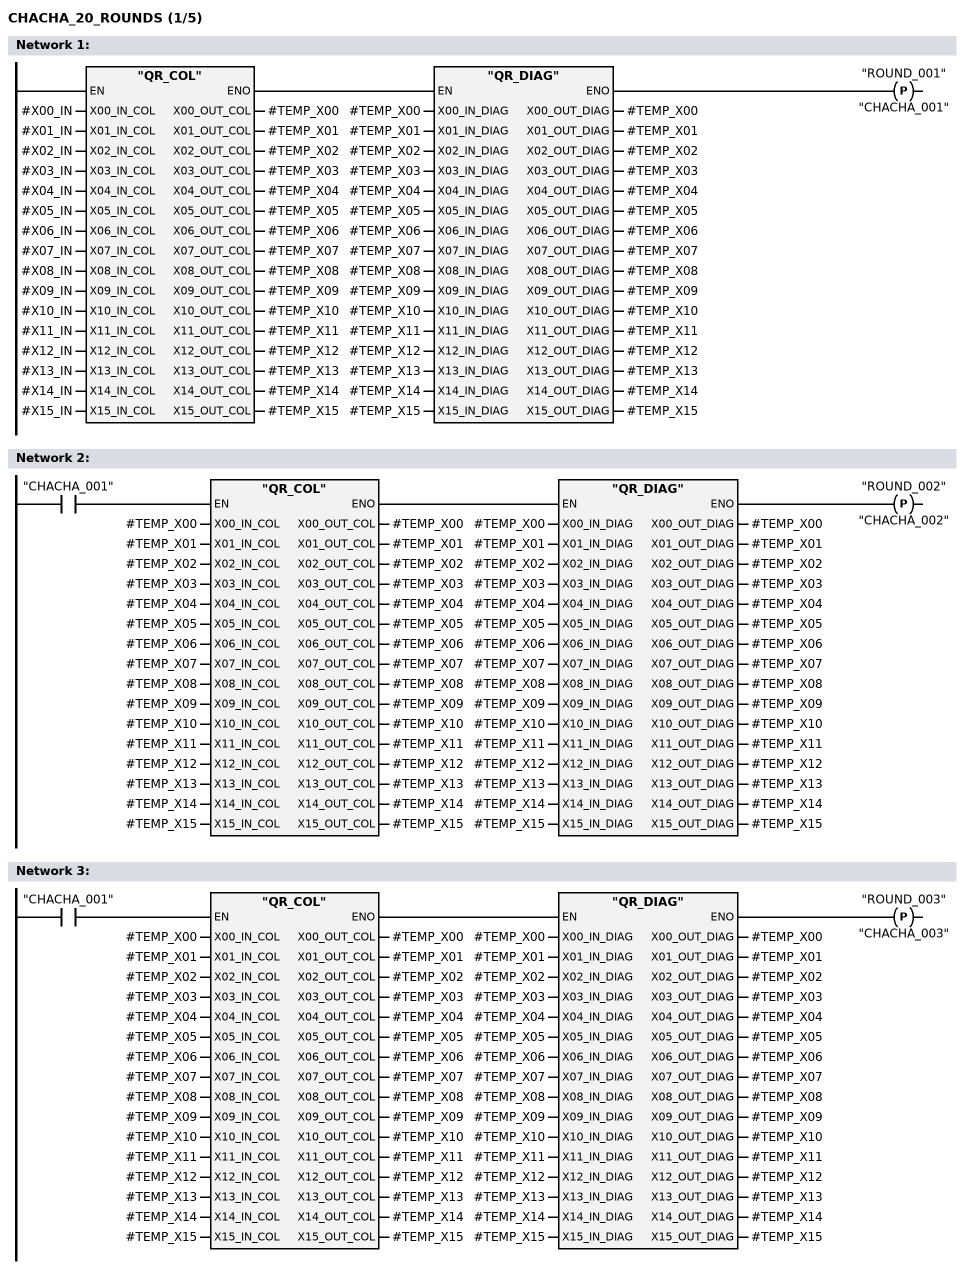
   "QR_COL"(X00_IN_COL := #X00_IN,
            X01_IN_COL := #X01_IN,
            X02_IN_COL := #X02_IN,
            X03_IN_COL := #X03_IN,
            X04_IN_COL := #X04_IN,
            X05_IN_COL := #X05_IN,
            X06_IN_COL := #X06_IN,
            X07_IN_COL := #X07_IN,
            X08_IN_COL := #X08_IN,
            X09_IN_COL := #X09_IN,
            X10_IN_COL := #X10_IN,
            X11_IN_COL := #X11_IN,
            X12_IN_COL := #X12_IN,
            X13_IN_COL := #X13_IN,
            X14_IN_COL := #X14_IN,
            X15_IN_COL := #X15_IN,
            X00_OUT_COL => #TEMP_X00,
            X01_OUT_COL => #TEMP_X01,
            X02_OUT_COL => #TEMP_X02,
            X03_OUT_COL => #TEMP_X03,
            X04_OUT_COL => #TEMP_X04,
            X05_OUT_COL => #TEMP_X05,
            X06_OUT_COL => #TEMP_X06,
            X07_OUT_COL => #TEMP_X07,
            X08_OUT_COL => #TEMP_X08,
            X09_OUT_COL => #TEMP_X09,
            X10_OUT_COL => #TEMP_X10,
            X11_OUT_COL => #TEMP_X11,
            X12_OUT_COL => #TEMP_X12,
            X13_OUT_COL => #TEMP_X13,
            X14_OUT_COL => #TEMP_X14,
            X15_OUT_COL => #TEMP_X15,
            ENO => #_w1);
   "QR_DIAG"(EN := #_w1,
             X00_IN_DIAG := #TEMP_X00,
             X01_IN_DIAG := #TEMP_X01,
             X02_IN_DIAG := #TEMP_X02,
             X03_IN_DIAG := #TEMP_X03,
             X04_IN_DIAG := #TEMP_X04,
             X05_IN_DIAG := #TEMP_X05,
             X06_IN_DIAG := #TEMP_X06,
             X07_IN_DIAG := #TEMP_X07,
             X08_IN_DIAG := #TEMP_X08,
             X09_IN_DIAG := #TEMP_X09,
             X10_IN_DIAG := #TEMP_X10,
             X11_IN_DIAG := #TEMP_X11,
             X12_IN_DIAG := #TEMP_X12,
             X13_IN_DIAG := #TEMP_X13,
             X14_IN_DIAG := #TEMP_X14,
             X15_IN_DIAG := #TEMP_X15,
             X00_OUT_DIAG => #TEMP_X00,
             X01_OUT_DIAG => #TEMP_X01,
             X02_OUT_DIAG => #TEMP_X02,
             X03_OUT_DIAG => #TEMP_X03,
             X04_OUT_DIAG => #TEMP_X04,
             X05_OUT_DIAG => #TEMP_X05,
             X06_OUT_DIAG => #TEMP_X06,
             X07_OUT_DIAG => #TEMP_X07,
             X08_OUT_DIAG => #TEMP_X08,
             X09_OUT_DIAG => #TEMP_X09,
             X10_OUT_DIAG => #TEMP_X10,
             X11_OUT_DIAG => #TEMP_X11,
             X12_OUT_DIAG => #TEMP_X12,
             X13_OUT_DIAG => #TEMP_X13,
             X14_OUT_DIAG => #TEMP_X14,
             X15_OUT_DIAG => #TEMP_X15,
             ENO => #_w2);
   "ROUND_001" := #_w2 AND NOT "CHACHA_001";   // rising edge
   "CHACHA_001" := #_w2;
END_REGION

REGION Network 2
   "QR_COL"(EN := "CHACHA_001",
            X00_IN_COL := #TEMP_X00,
            X01_IN_COL := #TEMP_X01,
            X02_IN_COL := #TEMP_X02,
            X03_IN_COL := #TEMP_X03,
            X04_IN_COL := #TEMP_X04,
            X05_IN_COL := #TEMP_X05,
            X06_IN_COL := #TEMP_X06,
            X07_IN_COL := #TEMP_X07,
            X08_IN_COL := #TEMP_X08,
            X09_IN_COL := #TEMP_X09,
            X10_IN_COL := #TEMP_X10,
            X11_IN_COL := #TEMP_X11,
            X12_IN_COL := #TEMP_X12,
            X13_IN_COL := #TEMP_X13,
            X14_IN_COL := #TEMP_X14,
            X15_IN_COL := #TEMP_X15,
            X00_OUT_COL => #TEMP_X00,
            X01_OUT_COL => #TEMP_X01,
            X02_OUT_COL => #TEMP_X02,
            X03_OUT_COL => #TEMP_X03,
            X04_OUT_COL => #TEMP_X04,
            X05_OUT_COL => #TEMP_X05,
            X06_OUT_COL => #TEMP_X06,
            X07_OUT_COL => #TEMP_X07,
            X08_OUT_COL => #TEMP_X08,
            X09_OUT_COL => #TEMP_X09,
            X10_OUT_COL => #TEMP_X10,
            X11_OUT_COL => #TEMP_X11,
            X12_OUT_COL => #TEMP_X12,
            X13_OUT_COL => #TEMP_X13,
            X14_OUT_COL => #TEMP_X14,
            X15_OUT_COL => #TEMP_X15,
            ENO => #_w1);
   "QR_DIAG"(EN := #_w1,
             X00_IN_DIAG := #TEMP_X00,
             X01_IN_DIAG := #TEMP_X01,
             X02_IN_DIAG := #TEMP_X02,
             X03_IN_DIAG := #TEMP_X03,
             X04_IN_DIAG := #TEMP_X04,
             X05_IN_DIAG := #TEMP_X05,
             X06_IN_DIAG := #TEMP_X06,
             X07_IN_DIAG := #TEMP_X07,
             X08_IN_DIAG := #TEMP_X08,
             X09_IN_DIAG := #TEMP_X09,
             X10_IN_DIAG := #TEMP_X10,
             X11_IN_DIAG := #TEMP_X11,
             X12_IN_DIAG := #TEMP_X12,
             X13_IN_DIAG := #TEMP_X13,
             X14_IN_DIAG := #TEMP_X14,
             X15_IN_DIAG := #TEMP_X15,
             X00_OUT_DIAG => #TEMP_X00,
             X01_OUT_DIAG => #TEMP_X01,
             X02_OUT_DIAG => #TEMP_X02,
             X03_OUT_DIAG => #TEMP_X03,
             X04_OUT_DIAG => #TEMP_X04,
             X05_OUT_DIAG => #TEMP_X05,
             X06_OUT_DIAG => #TEMP_X06,
             X07_OUT_DIAG => #TEMP_X07,
             X08_OUT_DIAG => #TEMP_X08,
             X09_OUT_DIAG => #TEMP_X09,
             X10_OUT_DIAG => #TEMP_X10,
             X11_OUT_DIAG => #TEMP_X11,
             X12_OUT_DIAG => #TEMP_X12,
             X13_OUT_DIAG => #TEMP_X13,
             X14_OUT_DIAG => #TEMP_X14,
             X15_OUT_DIAG => #TEMP_X15,
             ENO => #_w2);
   "ROUND_002" := #_w2 AND NOT "CHACHA_002";   // rising edge
   "CHACHA_002" := #_w2;
END_REGION

REGION Network 3
   "QR_COL"(EN := "CHACHA_001",
            X00_IN_COL := #TEMP_X00,
            X01_IN_COL := #TEMP_X01,
            X02_IN_COL := #TEMP_X02,
            X03_IN_COL := #TEMP_X03,
            X04_IN_COL := #TEMP_X04,
            X05_IN_COL := #TEMP_X05,
            X06_IN_COL := #TEMP_X06,
            X07_IN_COL := #TEMP_X07,
            X08_IN_COL := #TEMP_X08,
            X09_IN_COL := #TEMP_X09,
            X10_IN_COL := #TEMP_X10,
            X11_IN_COL := #TEMP_X11,
            X12_IN_COL := #TEMP_X12,
            X13_IN_COL := #TEMP_X13,
            X14_IN_COL := #TEMP_X14,
            X15_IN_COL := #TEMP_X15,
            X00_OUT_COL => #TEMP_X00,
            X01_OUT_COL => #TEMP_X01,
            X02_OUT_COL => #TEMP_X02,
            X03_OUT_COL => #TEMP_X03,
            X04_OUT_COL => #TEMP_X04,
            X05_OUT_COL => #TEMP_X05,
            X06_OUT_COL => #TEMP_X06,
            X07_OUT_COL => #TEMP_X07,
            X08_OUT_COL => #TEMP_X08,
            X09_OUT_COL => #TEMP_X09,
            X10_OUT_COL => #TEMP_X10,
            X11_OUT_COL => #TEMP_X11,
            X12_OUT_COL => #TEMP_X12,
            X13_OUT_COL => #TEMP_X13,
            X14_OUT_COL => #TEMP_X14,
            X15_OUT_COL => #TEMP_X15,
            ENO => #_w1);
   "QR_DIAG"(EN := #_w1,
             X00_IN_DIAG := #TEMP_X00,
             X01_IN_DIAG := #TEMP_X01,
             X02_IN_DIAG := #TEMP_X02,
             X03_IN_DIAG := #TEMP_X03,
             X04_IN_DIAG := #TEMP_X04,
             X05_IN_DIAG := #TEMP_X05,
             X06_IN_DIAG := #TEMP_X06,
             X07_IN_DIAG := #TEMP_X07,
             X08_IN_DIAG := #TEMP_X08,
             X09_IN_DIAG := #TEMP_X09,
             X10_IN_DIAG := #TEMP_X10,
             X11_IN_DIAG := #TEMP_X11,
             X12_IN_DIAG := #TEMP_X12,
             X13_IN_DIAG := #TEMP_X13,
             X14_IN_DIAG := #TEMP_X14,
             X15_IN_DIAG := #TEMP_X15,
             X00_OUT_DIAG => #TEMP_X00,
             X01_OUT_DIAG => #TEMP_X01,
             X02_OUT_DIAG => #TEMP_X02,
             X03_OUT_DIAG => #TEMP_X03,
             X04_OUT_DIAG => #TEMP_X04,
             X05_OUT_DIAG => #TEMP_X05,
             X06_OUT_DIAG => #TEMP_X06,
             X07_OUT_DIAG => #TEMP_X07,
             X08_OUT_DIAG => #TEMP_X08,
             X09_OUT_DIAG => #TEMP_X09,
             X10_OUT_DIAG => #TEMP_X10,
             X11_OUT_DIAG => #TEMP_X11,
             X12_OUT_DIAG => #TEMP_X12,
             X13_OUT_DIAG => #TEMP_X13,
             X14_OUT_DIAG => #TEMP_X14,
             X15_OUT_DIAG => #TEMP_X15,
             ENO => #_w2);
   "ROUND_003" := #_w2 AND NOT "CHACHA_003";   // rising edge
   "CHACHA_003" := #_w2;
END_REGION

REGION Network 4
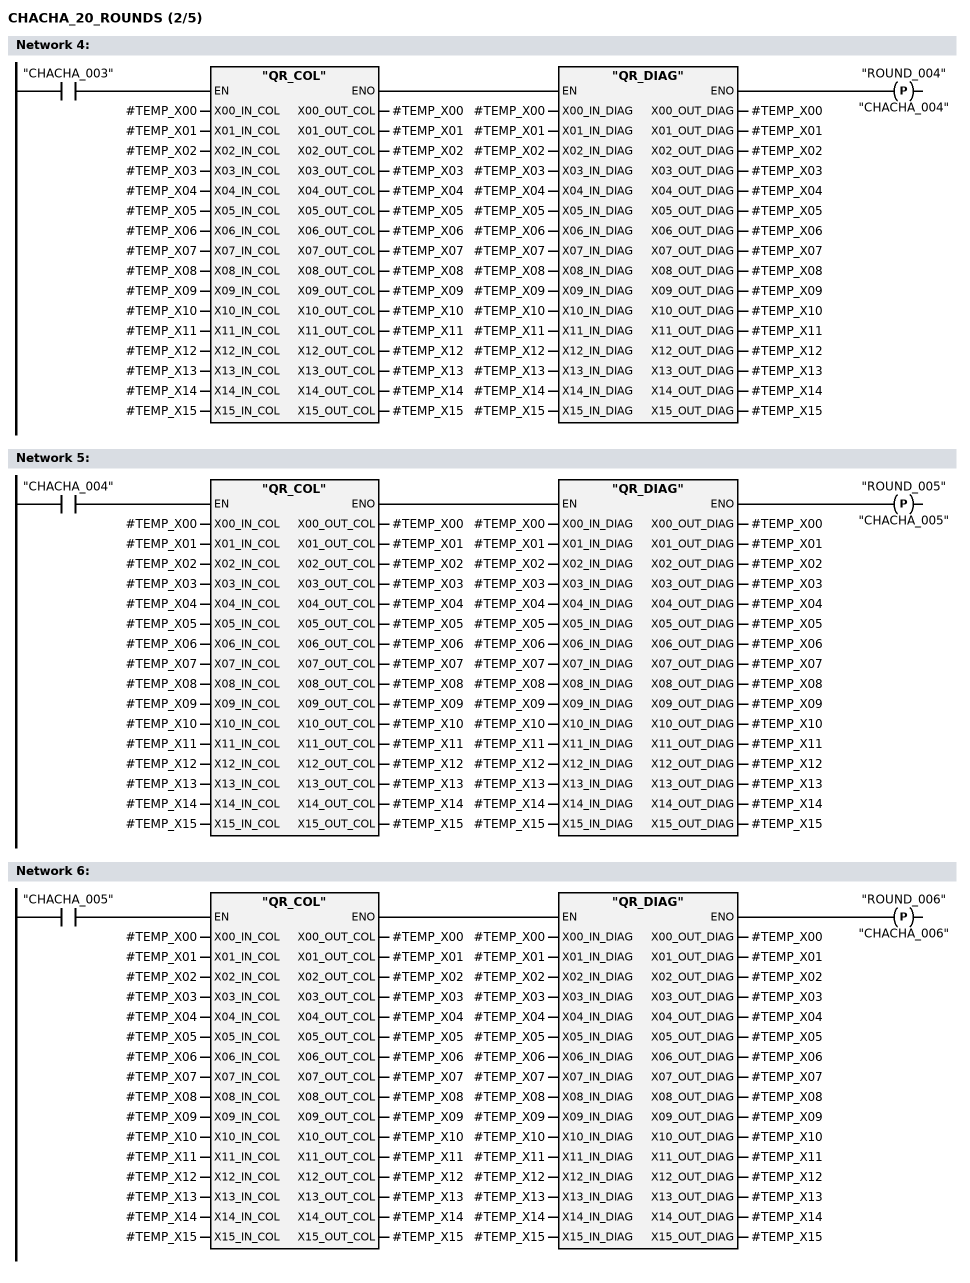
   "QR_COL"(EN := "CHACHA_003",
            X00_IN_COL := #TEMP_X00,
            X01_IN_COL := #TEMP_X01,
            X02_IN_COL := #TEMP_X02,
            X03_IN_COL := #TEMP_X03,
            X04_IN_COL := #TEMP_X04,
            X05_IN_COL := #TEMP_X05,
            X06_IN_COL := #TEMP_X06,
            X07_IN_COL := #TEMP_X07,
            X08_IN_COL := #TEMP_X08,
            X09_IN_COL := #TEMP_X09,
            X10_IN_COL := #TEMP_X10,
            X11_IN_COL := #TEMP_X11,
            X12_IN_COL := #TEMP_X12,
            X13_IN_COL := #TEMP_X13,
            X14_IN_COL := #TEMP_X14,
            X15_IN_COL := #TEMP_X15,
            X00_OUT_COL => #TEMP_X00,
            X01_OUT_COL => #TEMP_X01,
            X02_OUT_COL => #TEMP_X02,
            X03_OUT_COL => #TEMP_X03,
            X04_OUT_COL => #TEMP_X04,
            X05_OUT_COL => #TEMP_X05,
            X06_OUT_COL => #TEMP_X06,
            X07_OUT_COL => #TEMP_X07,
            X08_OUT_COL => #TEMP_X08,
            X09_OUT_COL => #TEMP_X09,
            X10_OUT_COL => #TEMP_X10,
            X11_OUT_COL => #TEMP_X11,
            X12_OUT_COL => #TEMP_X12,
            X13_OUT_COL => #TEMP_X13,
            X14_OUT_COL => #TEMP_X14,
            X15_OUT_COL => #TEMP_X15,
            ENO => #_w1);
   "QR_DIAG"(EN := #_w1,
             X00_IN_DIAG := #TEMP_X00,
             X01_IN_DIAG := #TEMP_X01,
             X02_IN_DIAG := #TEMP_X02,
             X03_IN_DIAG := #TEMP_X03,
             X04_IN_DIAG := #TEMP_X04,
             X05_IN_DIAG := #TEMP_X05,
             X06_IN_DIAG := #TEMP_X06,
             X07_IN_DIAG := #TEMP_X07,
             X08_IN_DIAG := #TEMP_X08,
             X09_IN_DIAG := #TEMP_X09,
             X10_IN_DIAG := #TEMP_X10,
             X11_IN_DIAG := #TEMP_X11,
             X12_IN_DIAG := #TEMP_X12,
             X13_IN_DIAG := #TEMP_X13,
             X14_IN_DIAG := #TEMP_X14,
             X15_IN_DIAG := #TEMP_X15,
             X00_OUT_DIAG => #TEMP_X00,
             X01_OUT_DIAG => #TEMP_X01,
             X02_OUT_DIAG => #TEMP_X02,
             X03_OUT_DIAG => #TEMP_X03,
             X04_OUT_DIAG => #TEMP_X04,
             X05_OUT_DIAG => #TEMP_X05,
             X06_OUT_DIAG => #TEMP_X06,
             X07_OUT_DIAG => #TEMP_X07,
             X08_OUT_DIAG => #TEMP_X08,
             X09_OUT_DIAG => #TEMP_X09,
             X10_OUT_DIAG => #TEMP_X10,
             X11_OUT_DIAG => #TEMP_X11,
             X12_OUT_DIAG => #TEMP_X12,
             X13_OUT_DIAG => #TEMP_X13,
             X14_OUT_DIAG => #TEMP_X14,
             X15_OUT_DIAG => #TEMP_X15,
             ENO => #_w2);
   "ROUND_004" := #_w2 AND NOT "CHACHA_004";   // rising edge
   "CHACHA_004" := #_w2;
END_REGION

REGION Network 5
   "QR_COL"(EN := "CHACHA_004",
            X00_IN_COL := #TEMP_X00,
            X01_IN_COL := #TEMP_X01,
            X02_IN_COL := #TEMP_X02,
            X03_IN_COL := #TEMP_X03,
            X04_IN_COL := #TEMP_X04,
            X05_IN_COL := #TEMP_X05,
            X06_IN_COL := #TEMP_X06,
            X07_IN_COL := #TEMP_X07,
            X08_IN_COL := #TEMP_X08,
            X09_IN_COL := #TEMP_X09,
            X10_IN_COL := #TEMP_X10,
            X11_IN_COL := #TEMP_X11,
            X12_IN_COL := #TEMP_X12,
            X13_IN_COL := #TEMP_X13,
            X14_IN_COL := #TEMP_X14,
            X15_IN_COL := #TEMP_X15,
            X00_OUT_COL => #TEMP_X00,
            X01_OUT_COL => #TEMP_X01,
            X02_OUT_COL => #TEMP_X02,
            X03_OUT_COL => #TEMP_X03,
            X04_OUT_COL => #TEMP_X04,
            X05_OUT_COL => #TEMP_X05,
            X06_OUT_COL => #TEMP_X06,
            X07_OUT_COL => #TEMP_X07,
            X08_OUT_COL => #TEMP_X08,
            X09_OUT_COL => #TEMP_X09,
            X10_OUT_COL => #TEMP_X10,
            X11_OUT_COL => #TEMP_X11,
            X12_OUT_COL => #TEMP_X12,
            X13_OUT_COL => #TEMP_X13,
            X14_OUT_COL => #TEMP_X14,
            X15_OUT_COL => #TEMP_X15,
            ENO => #_w1);
   "QR_DIAG"(EN := #_w1,
             X00_IN_DIAG := #TEMP_X00,
             X01_IN_DIAG := #TEMP_X01,
             X02_IN_DIAG := #TEMP_X02,
             X03_IN_DIAG := #TEMP_X03,
             X04_IN_DIAG := #TEMP_X04,
             X05_IN_DIAG := #TEMP_X05,
             X06_IN_DIAG := #TEMP_X06,
             X07_IN_DIAG := #TEMP_X07,
             X08_IN_DIAG := #TEMP_X08,
             X09_IN_DIAG := #TEMP_X09,
             X10_IN_DIAG := #TEMP_X10,
             X11_IN_DIAG := #TEMP_X11,
             X12_IN_DIAG := #TEMP_X12,
             X13_IN_DIAG := #TEMP_X13,
             X14_IN_DIAG := #TEMP_X14,
             X15_IN_DIAG := #TEMP_X15,
             X00_OUT_DIAG => #TEMP_X00,
             X01_OUT_DIAG => #TEMP_X01,
             X02_OUT_DIAG => #TEMP_X02,
             X03_OUT_DIAG => #TEMP_X03,
             X04_OUT_DIAG => #TEMP_X04,
             X05_OUT_DIAG => #TEMP_X05,
             X06_OUT_DIAG => #TEMP_X06,
             X07_OUT_DIAG => #TEMP_X07,
             X08_OUT_DIAG => #TEMP_X08,
             X09_OUT_DIAG => #TEMP_X09,
             X10_OUT_DIAG => #TEMP_X10,
             X11_OUT_DIAG => #TEMP_X11,
             X12_OUT_DIAG => #TEMP_X12,
             X13_OUT_DIAG => #TEMP_X13,
             X14_OUT_DIAG => #TEMP_X14,
             X15_OUT_DIAG => #TEMP_X15,
             ENO => #_w2);
   "ROUND_005" := #_w2 AND NOT "CHACHA_005";   // rising edge
   "CHACHA_005" := #_w2;
END_REGION

REGION Network 6
   "QR_COL"(EN := "CHACHA_005",
            X00_IN_COL := #TEMP_X00,
            X01_IN_COL := #TEMP_X01,
            X02_IN_COL := #TEMP_X02,
            X03_IN_COL := #TEMP_X03,
            X04_IN_COL := #TEMP_X04,
            X05_IN_COL := #TEMP_X05,
            X06_IN_COL := #TEMP_X06,
            X07_IN_COL := #TEMP_X07,
            X08_IN_COL := #TEMP_X08,
            X09_IN_COL := #TEMP_X09,
            X10_IN_COL := #TEMP_X10,
            X11_IN_COL := #TEMP_X11,
            X12_IN_COL := #TEMP_X12,
            X13_IN_COL := #TEMP_X13,
            X14_IN_COL := #TEMP_X14,
            X15_IN_COL := #TEMP_X15,
            X00_OUT_COL => #TEMP_X00,
            X01_OUT_COL => #TEMP_X01,
            X02_OUT_COL => #TEMP_X02,
            X03_OUT_COL => #TEMP_X03,
            X04_OUT_COL => #TEMP_X04,
            X05_OUT_COL => #TEMP_X05,
            X06_OUT_COL => #TEMP_X06,
            X07_OUT_COL => #TEMP_X07,
            X08_OUT_COL => #TEMP_X08,
            X09_OUT_COL => #TEMP_X09,
            X10_OUT_COL => #TEMP_X10,
            X11_OUT_COL => #TEMP_X11,
            X12_OUT_COL => #TEMP_X12,
            X13_OUT_COL => #TEMP_X13,
            X14_OUT_COL => #TEMP_X14,
            X15_OUT_COL => #TEMP_X15,
            ENO => #_w1);
   "QR_DIAG"(EN := #_w1,
             X00_IN_DIAG := #TEMP_X00,
             X01_IN_DIAG := #TEMP_X01,
             X02_IN_DIAG := #TEMP_X02,
             X03_IN_DIAG := #TEMP_X03,
             X04_IN_DIAG := #TEMP_X04,
             X05_IN_DIAG := #TEMP_X05,
             X06_IN_DIAG := #TEMP_X06,
             X07_IN_DIAG := #TEMP_X07,
             X08_IN_DIAG := #TEMP_X08,
             X09_IN_DIAG := #TEMP_X09,
             X10_IN_DIAG := #TEMP_X10,
             X11_IN_DIAG := #TEMP_X11,
             X12_IN_DIAG := #TEMP_X12,
             X13_IN_DIAG := #TEMP_X13,
             X14_IN_DIAG := #TEMP_X14,
             X15_IN_DIAG := #TEMP_X15,
             X00_OUT_DIAG => #TEMP_X00,
             X01_OUT_DIAG => #TEMP_X01,
             X02_OUT_DIAG => #TEMP_X02,
             X03_OUT_DIAG => #TEMP_X03,
             X04_OUT_DIAG => #TEMP_X04,
             X05_OUT_DIAG => #TEMP_X05,
             X06_OUT_DIAG => #TEMP_X06,
             X07_OUT_DIAG => #TEMP_X07,
             X08_OUT_DIAG => #TEMP_X08,
             X09_OUT_DIAG => #TEMP_X09,
             X10_OUT_DIAG => #TEMP_X10,
             X11_OUT_DIAG => #TEMP_X11,
             X12_OUT_DIAG => #TEMP_X12,
             X13_OUT_DIAG => #TEMP_X13,
             X14_OUT_DIAG => #TEMP_X14,
             X15_OUT_DIAG => #TEMP_X15,
             ENO => #_w2);
   "ROUND_006" := #_w2 AND NOT "CHACHA_006";   // rising edge
   "CHACHA_006" := #_w2;
END_REGION

REGION Network 7
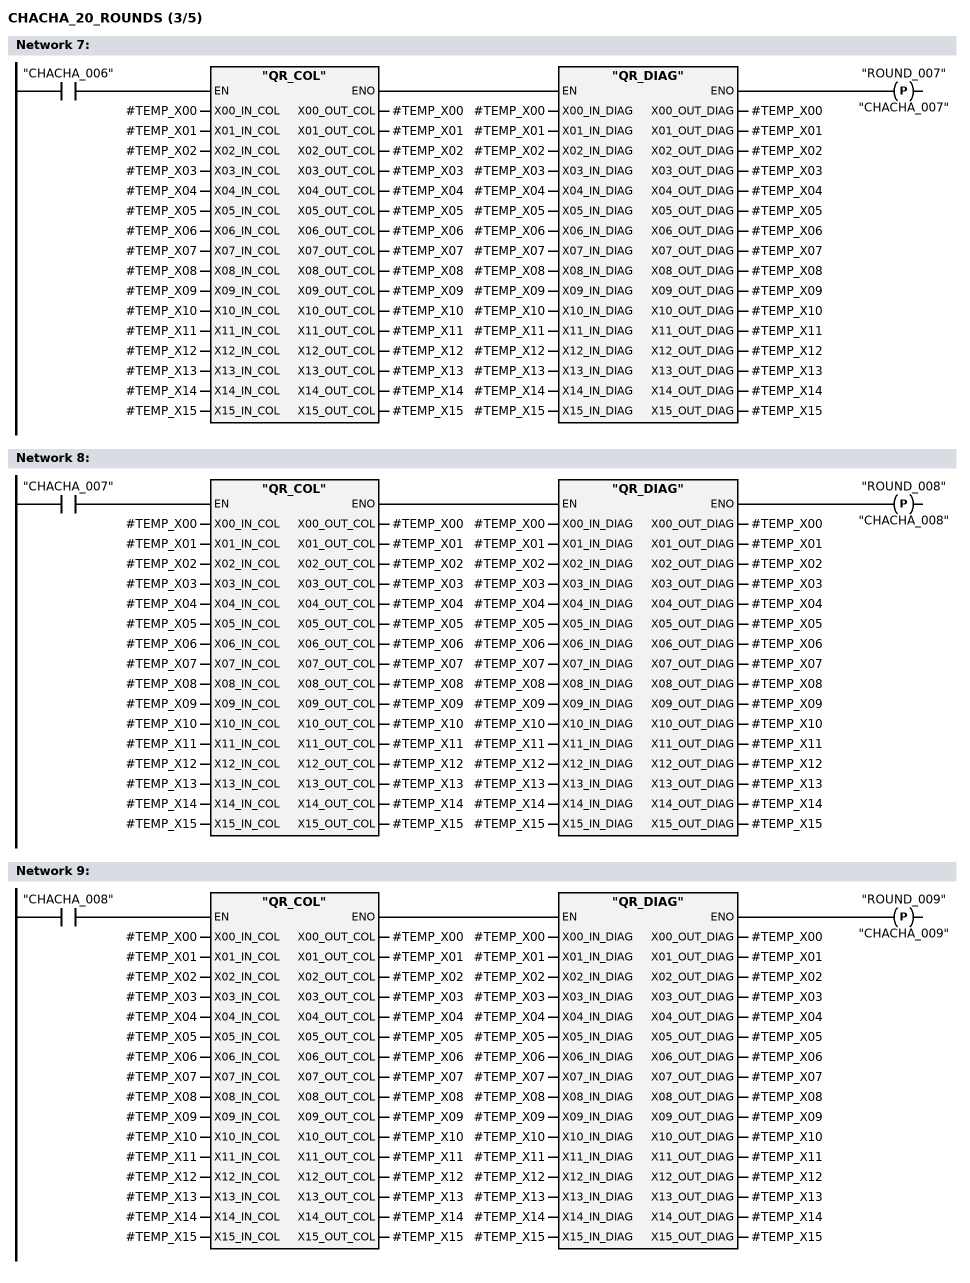
   "QR_COL"(EN := "CHACHA_006",
            X00_IN_COL := #TEMP_X00,
            X01_IN_COL := #TEMP_X01,
            X02_IN_COL := #TEMP_X02,
            X03_IN_COL := #TEMP_X03,
            X04_IN_COL := #TEMP_X04,
            X05_IN_COL := #TEMP_X05,
            X06_IN_COL := #TEMP_X06,
            X07_IN_COL := #TEMP_X07,
            X08_IN_COL := #TEMP_X08,
            X09_IN_COL := #TEMP_X09,
            X10_IN_COL := #TEMP_X10,
            X11_IN_COL := #TEMP_X11,
            X12_IN_COL := #TEMP_X12,
            X13_IN_COL := #TEMP_X13,
            X14_IN_COL := #TEMP_X14,
            X15_IN_COL := #TEMP_X15,
            X00_OUT_COL => #TEMP_X00,
            X01_OUT_COL => #TEMP_X01,
            X02_OUT_COL => #TEMP_X02,
            X03_OUT_COL => #TEMP_X03,
            X04_OUT_COL => #TEMP_X04,
            X05_OUT_COL => #TEMP_X05,
            X06_OUT_COL => #TEMP_X06,
            X07_OUT_COL => #TEMP_X07,
            X08_OUT_COL => #TEMP_X08,
            X09_OUT_COL => #TEMP_X09,
            X10_OUT_COL => #TEMP_X10,
            X11_OUT_COL => #TEMP_X11,
            X12_OUT_COL => #TEMP_X12,
            X13_OUT_COL => #TEMP_X13,
            X14_OUT_COL => #TEMP_X14,
            X15_OUT_COL => #TEMP_X15,
            ENO => #_w1);
   "QR_DIAG"(EN := #_w1,
             X00_IN_DIAG := #TEMP_X00,
             X01_IN_DIAG := #TEMP_X01,
             X02_IN_DIAG := #TEMP_X02,
             X03_IN_DIAG := #TEMP_X03,
             X04_IN_DIAG := #TEMP_X04,
             X05_IN_DIAG := #TEMP_X05,
             X06_IN_DIAG := #TEMP_X06,
             X07_IN_DIAG := #TEMP_X07,
             X08_IN_DIAG := #TEMP_X08,
             X09_IN_DIAG := #TEMP_X09,
             X10_IN_DIAG := #TEMP_X10,
             X11_IN_DIAG := #TEMP_X11,
             X12_IN_DIAG := #TEMP_X12,
             X13_IN_DIAG := #TEMP_X13,
             X14_IN_DIAG := #TEMP_X14,
             X15_IN_DIAG := #TEMP_X15,
             X00_OUT_DIAG => #TEMP_X00,
             X01_OUT_DIAG => #TEMP_X01,
             X02_OUT_DIAG => #TEMP_X02,
             X03_OUT_DIAG => #TEMP_X03,
             X04_OUT_DIAG => #TEMP_X04,
             X05_OUT_DIAG => #TEMP_X05,
             X06_OUT_DIAG => #TEMP_X06,
             X07_OUT_DIAG => #TEMP_X07,
             X08_OUT_DIAG => #TEMP_X08,
             X09_OUT_DIAG => #TEMP_X09,
             X10_OUT_DIAG => #TEMP_X10,
             X11_OUT_DIAG => #TEMP_X11,
             X12_OUT_DIAG => #TEMP_X12,
             X13_OUT_DIAG => #TEMP_X13,
             X14_OUT_DIAG => #TEMP_X14,
             X15_OUT_DIAG => #TEMP_X15,
             ENO => #_w2);
   "ROUND_007" := #_w2 AND NOT "CHACHA_007";   // rising edge
   "CHACHA_007" := #_w2;
END_REGION

REGION Network 8
   "QR_COL"(EN := "CHACHA_007",
            X00_IN_COL := #TEMP_X00,
            X01_IN_COL := #TEMP_X01,
            X02_IN_COL := #TEMP_X02,
            X03_IN_COL := #TEMP_X03,
            X04_IN_COL := #TEMP_X04,
            X05_IN_COL := #TEMP_X05,
            X06_IN_COL := #TEMP_X06,
            X07_IN_COL := #TEMP_X07,
            X08_IN_COL := #TEMP_X08,
            X09_IN_COL := #TEMP_X09,
            X10_IN_COL := #TEMP_X10,
            X11_IN_COL := #TEMP_X11,
            X12_IN_COL := #TEMP_X12,
            X13_IN_COL := #TEMP_X13,
            X14_IN_COL := #TEMP_X14,
            X15_IN_COL := #TEMP_X15,
            X00_OUT_COL => #TEMP_X00,
            X01_OUT_COL => #TEMP_X01,
            X02_OUT_COL => #TEMP_X02,
            X03_OUT_COL => #TEMP_X03,
            X04_OUT_COL => #TEMP_X04,
            X05_OUT_COL => #TEMP_X05,
            X06_OUT_COL => #TEMP_X06,
            X07_OUT_COL => #TEMP_X07,
            X08_OUT_COL => #TEMP_X08,
            X09_OUT_COL => #TEMP_X09,
            X10_OUT_COL => #TEMP_X10,
            X11_OUT_COL => #TEMP_X11,
            X12_OUT_COL => #TEMP_X12,
            X13_OUT_COL => #TEMP_X13,
            X14_OUT_COL => #TEMP_X14,
            X15_OUT_COL => #TEMP_X15,
            ENO => #_w1);
   "QR_DIAG"(EN := #_w1,
             X00_IN_DIAG := #TEMP_X00,
             X01_IN_DIAG := #TEMP_X01,
             X02_IN_DIAG := #TEMP_X02,
             X03_IN_DIAG := #TEMP_X03,
             X04_IN_DIAG := #TEMP_X04,
             X05_IN_DIAG := #TEMP_X05,
             X06_IN_DIAG := #TEMP_X06,
             X07_IN_DIAG := #TEMP_X07,
             X08_IN_DIAG := #TEMP_X08,
             X09_IN_DIAG := #TEMP_X09,
             X10_IN_DIAG := #TEMP_X10,
             X11_IN_DIAG := #TEMP_X11,
             X12_IN_DIAG := #TEMP_X12,
             X13_IN_DIAG := #TEMP_X13,
             X14_IN_DIAG := #TEMP_X14,
             X15_IN_DIAG := #TEMP_X15,
             X00_OUT_DIAG => #TEMP_X00,
             X01_OUT_DIAG => #TEMP_X01,
             X02_OUT_DIAG => #TEMP_X02,
             X03_OUT_DIAG => #TEMP_X03,
             X04_OUT_DIAG => #TEMP_X04,
             X05_OUT_DIAG => #TEMP_X05,
             X06_OUT_DIAG => #TEMP_X06,
             X07_OUT_DIAG => #TEMP_X07,
             X08_OUT_DIAG => #TEMP_X08,
             X09_OUT_DIAG => #TEMP_X09,
             X10_OUT_DIAG => #TEMP_X10,
             X11_OUT_DIAG => #TEMP_X11,
             X12_OUT_DIAG => #TEMP_X12,
             X13_OUT_DIAG => #TEMP_X13,
             X14_OUT_DIAG => #TEMP_X14,
             X15_OUT_DIAG => #TEMP_X15,
             ENO => #_w2);
   "ROUND_008" := #_w2 AND NOT "CHACHA_008";   // rising edge
   "CHACHA_008" := #_w2;
END_REGION

REGION Network 9
   "QR_COL"(EN := "CHACHA_008",
            X00_IN_COL := #TEMP_X00,
            X01_IN_COL := #TEMP_X01,
            X02_IN_COL := #TEMP_X02,
            X03_IN_COL := #TEMP_X03,
            X04_IN_COL := #TEMP_X04,
            X05_IN_COL := #TEMP_X05,
            X06_IN_COL := #TEMP_X06,
            X07_IN_COL := #TEMP_X07,
            X08_IN_COL := #TEMP_X08,
            X09_IN_COL := #TEMP_X09,
            X10_IN_COL := #TEMP_X10,
            X11_IN_COL := #TEMP_X11,
            X12_IN_COL := #TEMP_X12,
            X13_IN_COL := #TEMP_X13,
            X14_IN_COL := #TEMP_X14,
            X15_IN_COL := #TEMP_X15,
            X00_OUT_COL => #TEMP_X00,
            X01_OUT_COL => #TEMP_X01,
            X02_OUT_COL => #TEMP_X02,
            X03_OUT_COL => #TEMP_X03,
            X04_OUT_COL => #TEMP_X04,
            X05_OUT_COL => #TEMP_X05,
            X06_OUT_COL => #TEMP_X06,
            X07_OUT_COL => #TEMP_X07,
            X08_OUT_COL => #TEMP_X08,
            X09_OUT_COL => #TEMP_X09,
            X10_OUT_COL => #TEMP_X10,
            X11_OUT_COL => #TEMP_X11,
            X12_OUT_COL => #TEMP_X12,
            X13_OUT_COL => #TEMP_X13,
            X14_OUT_COL => #TEMP_X14,
            X15_OUT_COL => #TEMP_X15,
            ENO => #_w1);
   "QR_DIAG"(EN := #_w1,
             X00_IN_DIAG := #TEMP_X00,
             X01_IN_DIAG := #TEMP_X01,
             X02_IN_DIAG := #TEMP_X02,
             X03_IN_DIAG := #TEMP_X03,
             X04_IN_DIAG := #TEMP_X04,
             X05_IN_DIAG := #TEMP_X05,
             X06_IN_DIAG := #TEMP_X06,
             X07_IN_DIAG := #TEMP_X07,
             X08_IN_DIAG := #TEMP_X08,
             X09_IN_DIAG := #TEMP_X09,
             X10_IN_DIAG := #TEMP_X10,
             X11_IN_DIAG := #TEMP_X11,
             X12_IN_DIAG := #TEMP_X12,
             X13_IN_DIAG := #TEMP_X13,
             X14_IN_DIAG := #TEMP_X14,
             X15_IN_DIAG := #TEMP_X15,
             X00_OUT_DIAG => #TEMP_X00,
             X01_OUT_DIAG => #TEMP_X01,
             X02_OUT_DIAG => #TEMP_X02,
             X03_OUT_DIAG => #TEMP_X03,
             X04_OUT_DIAG => #TEMP_X04,
             X05_OUT_DIAG => #TEMP_X05,
             X06_OUT_DIAG => #TEMP_X06,
             X07_OUT_DIAG => #TEMP_X07,
             X08_OUT_DIAG => #TEMP_X08,
             X09_OUT_DIAG => #TEMP_X09,
             X10_OUT_DIAG => #TEMP_X10,
             X11_OUT_DIAG => #TEMP_X11,
             X12_OUT_DIAG => #TEMP_X12,
             X13_OUT_DIAG => #TEMP_X13,
             X14_OUT_DIAG => #TEMP_X14,
             X15_OUT_DIAG => #TEMP_X15,
             ENO => #_w2);
   "ROUND_009" := #_w2 AND NOT "CHACHA_009";   // rising edge
   "CHACHA_009" := #_w2;
END_REGION

REGION Network 10
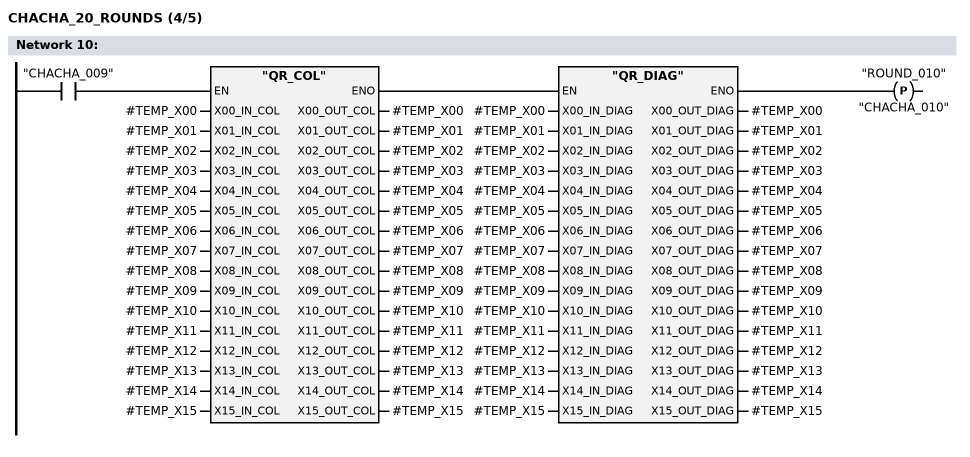
   "QR_COL"(EN := "CHACHA_009",
            X00_IN_COL := #TEMP_X00,
            X01_IN_COL := #TEMP_X01,
            X02_IN_COL := #TEMP_X02,
            X03_IN_COL := #TEMP_X03,
            X04_IN_COL := #TEMP_X04,
            X05_IN_COL := #TEMP_X05,
            X06_IN_COL := #TEMP_X06,
            X07_IN_COL := #TEMP_X07,
            X08_IN_COL := #TEMP_X08,
            X09_IN_COL := #TEMP_X09,
            X10_IN_COL := #TEMP_X10,
            X11_IN_COL := #TEMP_X11,
            X12_IN_COL := #TEMP_X12,
            X13_IN_COL := #TEMP_X13,
            X14_IN_COL := #TEMP_X14,
            X15_IN_COL := #TEMP_X15,
            X00_OUT_COL => #TEMP_X00,
            X01_OUT_COL => #TEMP_X01,
            X02_OUT_COL => #TEMP_X02,
            X03_OUT_COL => #TEMP_X03,
            X04_OUT_COL => #TEMP_X04,
            X05_OUT_COL => #TEMP_X05,
            X06_OUT_COL => #TEMP_X06,
            X07_OUT_COL => #TEMP_X07,
            X08_OUT_COL => #TEMP_X08,
            X09_OUT_COL => #TEMP_X09,
            X10_OUT_COL => #TEMP_X10,
            X11_OUT_COL => #TEMP_X11,
            X12_OUT_COL => #TEMP_X12,
            X13_OUT_COL => #TEMP_X13,
            X14_OUT_COL => #TEMP_X14,
            X15_OUT_COL => #TEMP_X15,
            ENO => #_w1);
   "QR_DIAG"(EN := #_w1,
             X00_IN_DIAG := #TEMP_X00,
             X01_IN_DIAG := #TEMP_X01,
             X02_IN_DIAG := #TEMP_X02,
             X03_IN_DIAG := #TEMP_X03,
             X04_IN_DIAG := #TEMP_X04,
             X05_IN_DIAG := #TEMP_X05,
             X06_IN_DIAG := #TEMP_X06,
             X07_IN_DIAG := #TEMP_X07,
             X08_IN_DIAG := #TEMP_X08,
             X09_IN_DIAG := #TEMP_X09,
             X10_IN_DIAG := #TEMP_X10,
             X11_IN_DIAG := #TEMP_X11,
             X12_IN_DIAG := #TEMP_X12,
             X13_IN_DIAG := #TEMP_X13,
             X14_IN_DIAG := #TEMP_X14,
             X15_IN_DIAG := #TEMP_X15,
             X00_OUT_DIAG => #TEMP_X00,
             X01_OUT_DIAG => #TEMP_X01,
             X02_OUT_DIAG => #TEMP_X02,
             X03_OUT_DIAG => #TEMP_X03,
             X04_OUT_DIAG => #TEMP_X04,
             X05_OUT_DIAG => #TEMP_X05,
             X06_OUT_DIAG => #TEMP_X06,
             X07_OUT_DIAG => #TEMP_X07,
             X08_OUT_DIAG => #TEMP_X08,
             X09_OUT_DIAG => #TEMP_X09,
             X10_OUT_DIAG => #TEMP_X10,
             X11_OUT_DIAG => #TEMP_X11,
             X12_OUT_DIAG => #TEMP_X12,
             X13_OUT_DIAG => #TEMP_X13,
             X14_OUT_DIAG => #TEMP_X14,
             X15_OUT_DIAG => #TEMP_X15,
             ENO => #_w2);
   "ROUND_010" := #_w2 AND NOT "CHACHA_010";   // rising edge
   "CHACHA_010" := #_w2;
END_REGION

REGION Network 11
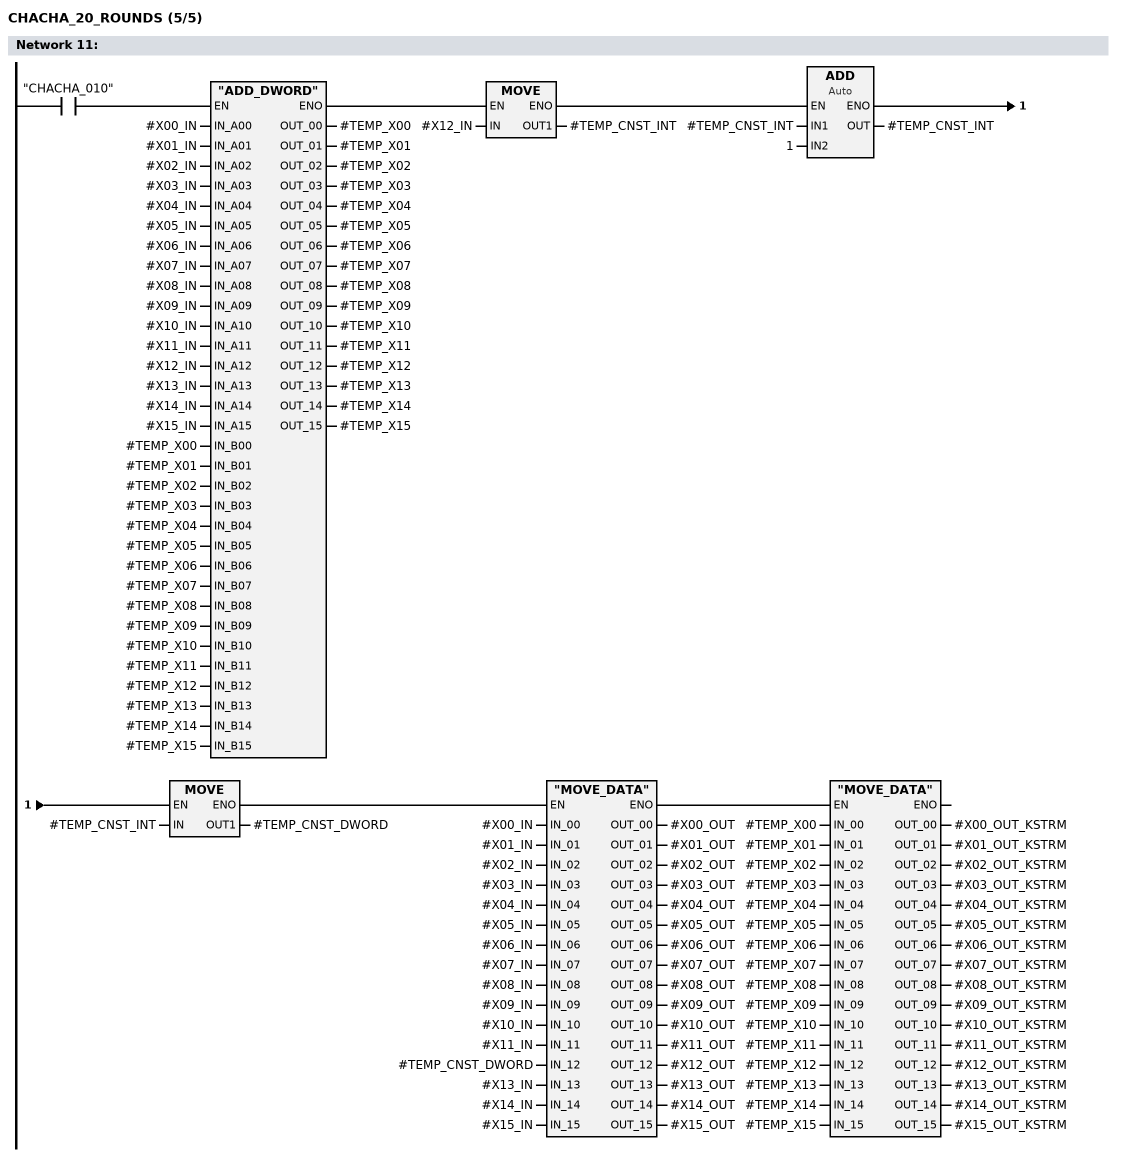
   RUNG wire#powerrail
      Contact( "CHACHA_010" )
      "ADD_DWORD"(IN_A00 := #X00_IN, IN_A01 := #X01_IN, IN_A02 := #X02_IN, IN_A03 := #X03_IN, IN_A04 := #X04_IN, IN_A05 := #X05_IN, IN_A06 := #X06_IN, IN_A07 := #X07_IN, IN_A08 := #X08_IN, IN_A09 := #X09_IN, IN_A10 := #X10_IN, IN_A11 := #X11_IN, IN_A12 := #X12_IN, IN_A13 := #X13_IN, IN_A14 := #X14_IN, IN_A15 := #X15_IN, IN_B00 := #TEMP_X00, IN_B01 := #TEMP_X01, IN_B02 := #TEMP_X02, IN_B03 := #TEMP_X03, IN_B04 := #TEMP_X04, IN_B05 := #TEMP_X05, IN_B06 := #TEMP_X06, IN_B07 := #TEMP_X07, IN_B08 := #TEMP_X08, IN_B09 := #TEMP_X09, IN_B10 := #TEMP_X10, IN_B11 := #TEMP_X11, IN_B12 := #TEMP_X12, IN_B13 := #TEMP_X13, IN_B14 := #TEMP_X14, IN_B15 := #TEMP_X15, OUT_00 => #TEMP_X00, OUT_01 => #TEMP_X01, OUT_02 => #TEMP_X02, OUT_03 => #TEMP_X03, OUT_04 => #TEMP_X04, OUT_05 => #TEMP_X05, OUT_06 => #TEMP_X06, OUT_07 => #TEMP_X07, OUT_08 => #TEMP_X08, OUT_09 => #TEMP_X09, OUT_10 => #TEMP_X10, OUT_11 => #TEMP_X11, OUT_12 => #TEMP_X12, OUT_13 => #TEMP_X13, OUT_14 => #TEMP_X14, OUT_15 => #TEMP_X15)
      { S7_GenerateENO := "TRUE" } Move(in := #X12_IN, out1 => #TEMP_CNST_INT)
      { S7_GenerateENO := "TRUE" } Add(in1 := #TEMP_CNST_INT, in2 := 1, out => #TEMP_CNST_INT)
      { S7_GenerateENO := "TRUE" } Move(in := #TEMP_CNST_INT, out1 => #TEMP_CNST_DWORD)
      "MOVE_DATA"(IN_00 := #X00_IN, IN_01 := #X01_IN, IN_02 := #X02_IN, IN_03 := #X03_IN, IN_04 := #X04_IN, IN_05 := #X05_IN, IN_06 := #X06_IN, IN_07 := #X07_IN, IN_08 := #X08_IN, IN_09 := #X09_IN, IN_10 := #X10_IN, IN_11 := #X11_IN, IN_12 := #TEMP_CNST_DWORD, IN_13 := #X13_IN, IN_14 := #X14_IN, IN_15 := #X15_IN, OUT_00 => #X00_OUT, OUT_01 => #X01_OUT, OUT_02 => #X02_OUT, OUT_03 => #X03_OUT, OUT_04 => #X04_OUT, OUT_05 => #X05_OUT, OUT_06 => #X06_OUT, OUT_07 => #X07_OUT, OUT_08 => #X08_OUT, OUT_09 => #X09_OUT, OUT_10 => #X10_OUT, OUT_11 => #X11_OUT, OUT_12 => #X12_OUT, OUT_13 => #X13_OUT, OUT_14 => #X14_OUT, OUT_15 => #X15_OUT)
      "MOVE_DATA"(IN_00 := #TEMP_X00, IN_01 := #TEMP_X01, IN_02 := #TEMP_X02, IN_03 := #TEMP_X03, IN_04 := #TEMP_X04, IN_05 := #TEMP_X05, IN_06 := #TEMP_X06, IN_07 := #TEMP_X07, IN_08 := #TEMP_X08, IN_09 := #TEMP_X09, IN_10 := #TEMP_X10, IN_11 := #TEMP_X11, IN_12 := #TEMP_X12, IN_13 := #TEMP_X13, IN_14 := #TEMP_X14, IN_15 := #TEMP_X15, OUT_00 => #X00_OUT_KSTRM, OUT_01 => #X01_OUT_KSTRM, OUT_02 => #X02_OUT_KSTRM, OUT_03 => #X03_OUT_KSTRM, OUT_04 => #X04_OUT_KSTRM, OUT_05 => #X05_OUT_KSTRM, OUT_06 => #X06_OUT_KSTRM, OUT_07 => #X07_OUT_KSTRM, OUT_08 => #X08_OUT_KSTRM, OUT_09 => #X09_OUT_KSTRM, OUT_10 => #X10_OUT_KSTRM, OUT_11 => #X11_OUT_KSTRM, OUT_12 => #X12_OUT_KSTRM, OUT_13 => #X13_OUT_KSTRM, OUT_14 => #X14_OUT_KSTRM, OUT_15 => #X15_OUT_KSTRM)
   END_RUNG
   RUNG wire#powerrail
   END_RUNG
   // the same network as SCL:
   // ENO of a box is taken as its EN; it also drops when the box reports an error
   "ADD_DWORD"(EN := "CHACHA_010",
               IN_A00 := #X00_IN,
               IN_A01 := #X01_IN,
               IN_A02 := #X02_IN,
               IN_A03 := #X03_IN,
               IN_A04 := #X04_IN,
               IN_A05 := #X05_IN,
               IN_A06 := #X06_IN,
               IN_A07 := #X07_IN,
               IN_A08 := #X08_IN,
               IN_A09 := #X09_IN,
               IN_A10 := #X10_IN,
               IN_A11 := #X11_IN,
               IN_A12 := #X12_IN,
               IN_A13 := #X13_IN,
               IN_A14 := #X14_IN,
               IN_A15 := #X15_IN,
               IN_B00 := #TEMP_X00,
               IN_B01 := #TEMP_X01,
               IN_B02 := #TEMP_X02,
               IN_B03 := #TEMP_X03,
               IN_B04 := #TEMP_X04,
               IN_B05 := #TEMP_X05,
               IN_B06 := #TEMP_X06,
               IN_B07 := #TEMP_X07,
               IN_B08 := #TEMP_X08,
               IN_B09 := #TEMP_X09,
               IN_B10 := #TEMP_X10,
               IN_B11 := #TEMP_X11,
               IN_B12 := #TEMP_X12,
               IN_B13 := #TEMP_X13,
               IN_B14 := #TEMP_X14,
               IN_B15 := #TEMP_X15,
               OUT_00 => #TEMP_X00,
               OUT_01 => #TEMP_X01,
               OUT_02 => #TEMP_X02,
               OUT_03 => #TEMP_X03,
               OUT_04 => #TEMP_X04,
               OUT_05 => #TEMP_X05,
               OUT_06 => #TEMP_X06,
               OUT_07 => #TEMP_X07,
               OUT_08 => #TEMP_X08,
               OUT_09 => #TEMP_X09,
               OUT_10 => #TEMP_X10,
               OUT_11 => #TEMP_X11,
               OUT_12 => #TEMP_X12,
               OUT_13 => #TEMP_X13,
               OUT_14 => #TEMP_X14,
               OUT_15 => #TEMP_X15,
               ENO => #_w1);
   IF #_w1 THEN
       #TEMP_CNST_INT := #X12_IN;
       #TEMP_CNST_INT := #TEMP_CNST_INT + 1;
       #TEMP_CNST_DWORD := #TEMP_CNST_INT;
   END_IF;
   "MOVE_DATA"(EN := #_w1,
               IN_00 := #X00_IN,
               IN_01 := #X01_IN,
               IN_02 := #X02_IN,
               IN_03 := #X03_IN,
               IN_04 := #X04_IN,
               IN_05 := #X05_IN,
               IN_06 := #X06_IN,
               IN_07 := #X07_IN,
               IN_08 := #X08_IN,
               IN_09 := #X09_IN,
               IN_10 := #X10_IN,
               IN_11 := #X11_IN,
               IN_12 := #TEMP_CNST_DWORD,
               IN_13 := #X13_IN,
               IN_14 := #X14_IN,
               IN_15 := #X15_IN,
               OUT_00 => #X00_OUT,
               OUT_01 => #X01_OUT,
               OUT_02 => #X02_OUT,
               OUT_03 => #X03_OUT,
               OUT_04 => #X04_OUT,
               OUT_05 => #X05_OUT,
               OUT_06 => #X06_OUT,
               OUT_07 => #X07_OUT,
               OUT_08 => #X08_OUT,
               OUT_09 => #X09_OUT,
               OUT_10 => #X10_OUT,
               OUT_11 => #X11_OUT,
               OUT_12 => #X12_OUT,
               OUT_13 => #X13_OUT,
               OUT_14 => #X14_OUT,
               OUT_15 => #X15_OUT,
               ENO => #_w2);
   IF #_w2 THEN
       "MOVE_DATA"(IN_00 := #TEMP_X00,
                   IN_01 := #TEMP_X01,
                   IN_02 := #TEMP_X02,
                   IN_03 := #TEMP_X03,
                   IN_04 := #TEMP_X04,
                   IN_05 := #TEMP_X05,
                   IN_06 := #TEMP_X06,
                   IN_07 := #TEMP_X07,
                   IN_08 := #TEMP_X08,
                   IN_09 := #TEMP_X09,
                   IN_10 := #TEMP_X10,
                   IN_11 := #TEMP_X11,
                   IN_12 := #TEMP_X12,
                   IN_13 := #TEMP_X13,
                   IN_14 := #TEMP_X14,
                   IN_15 := #TEMP_X15,
                   OUT_00 => #X00_OUT_KSTRM,
                   OUT_01 => #X01_OUT_KSTRM,
                   OUT_02 => #X02_OUT_KSTRM,
                   OUT_03 => #X03_OUT_KSTRM,
                   OUT_04 => #X04_OUT_KSTRM,
                   OUT_05 => #X05_OUT_KSTRM,
                   OUT_06 => #X06_OUT_KSTRM,
                   OUT_07 => #X07_OUT_KSTRM,
                   OUT_08 => #X08_OUT_KSTRM,
                   OUT_09 => #X09_OUT_KSTRM,
                   OUT_10 => #X10_OUT_KSTRM,
                   OUT_11 => #X11_OUT_KSTRM,
                   OUT_12 => #X12_OUT_KSTRM,
                   OUT_13 => #X13_OUT_KSTRM,
                   OUT_14 => #X14_OUT_KSTRM,
                   OUT_15 => #X15_OUT_KSTRM);
   END_IF;
END_REGION
END_FUNCTION

FUNCTION "CHACHA_1_ROUND" : Void   // FC6, LAD
{ S7_Optimized_Access := 'TRUE' }
VERSION : 0.1
   VAR_INPUT
      X00_IN : DWord;
      X01_IN : DWord;
      X02_IN : DWord;
      X03_IN : DWord;
      X04_IN : DWord;
      X05_IN : DWord;
      X06_IN : DWord;
      X07_IN : DWord;
      X08_IN : DWord;
      X09_IN : DWord;
      X10_IN : DWord;
      X11_IN : DWord;
      X12_IN : DWord;
      X13_IN : DWord;
      X14_IN : DWord;
      X15_IN : DWord;
   END_VAR
   VAR_OUTPUT
      X00_OUT : DWord;
      X01_OUT : DWord;
      X02_OUT : DWord;
      X03_OUT : DWord;
      X04_OUT : DWord;
      X05_OUT : DWord;
      X06_OUT : DWord;
      X07_OUT : DWord;
      X08_OUT : DWord;
      X09_OUT : DWord;
      X10_OUT : DWord;
      X11_OUT : DWord;
      X12_OUT : DWord;
      X13_OUT : DWord;
      X14_OUT : DWord;
      X15_OUT : DWord;
   END_VAR
   VAR_TEMP
      TEMP_X00 : DWord;
      TEMP_X01 : DWord;
      TEMP_X02 : DWord;
      TEMP_X03 : DWord;
      TEMP_X04 : DWord;
      TEMP_X05 : DWord;
      TEMP_X06 : DWord;
      TEMP_X07 : DWord;
      TEMP_X08 : DWord;
      TEMP_X09 : DWord;
      TEMP_X10 : DWord;
      TEMP_X11 : DWord;
      TEMP_X12 : DWord;
      TEMP_X13 : DWord;
      TEMP_X14 : DWord;
      TEMP_X15 : DWord;
   END_VAR
BEGIN

REGION Network 1
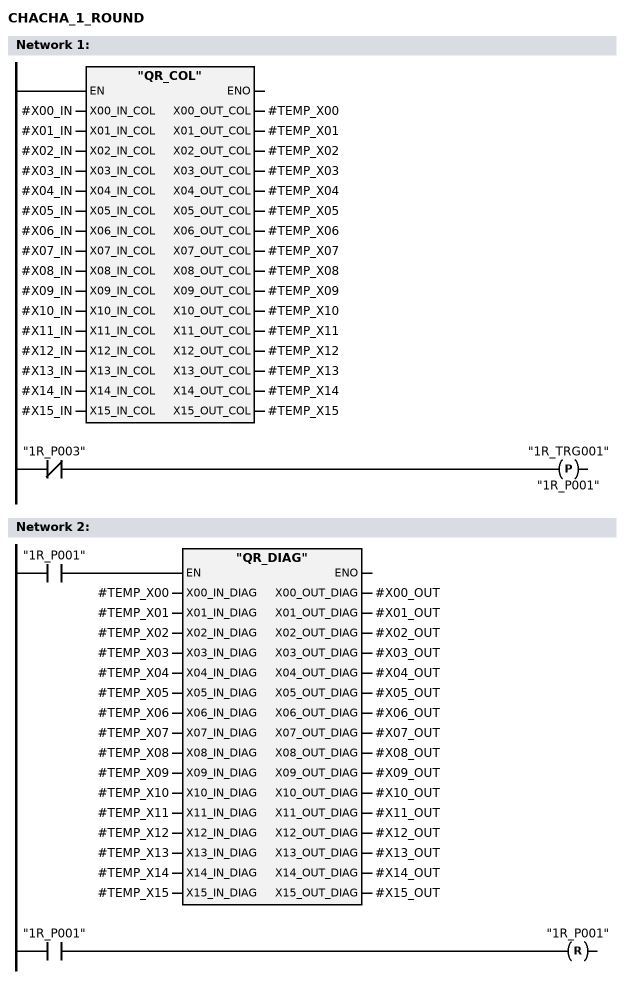
   "QR_COL"(X00_IN_COL := #X00_IN,
            X01_IN_COL := #X01_IN,
            X02_IN_COL := #X02_IN,
            X03_IN_COL := #X03_IN,
            X04_IN_COL := #X04_IN,
            X05_IN_COL := #X05_IN,
            X06_IN_COL := #X06_IN,
            X07_IN_COL := #X07_IN,
            X08_IN_COL := #X08_IN,
            X09_IN_COL := #X09_IN,
            X10_IN_COL := #X10_IN,
            X11_IN_COL := #X11_IN,
            X12_IN_COL := #X12_IN,
            X13_IN_COL := #X13_IN,
            X14_IN_COL := #X14_IN,
            X15_IN_COL := #X15_IN,
            X00_OUT_COL => #TEMP_X00,
            X01_OUT_COL => #TEMP_X01,
            X02_OUT_COL => #TEMP_X02,
            X03_OUT_COL => #TEMP_X03,
            X04_OUT_COL => #TEMP_X04,
            X05_OUT_COL => #TEMP_X05,
            X06_OUT_COL => #TEMP_X06,
            X07_OUT_COL => #TEMP_X07,
            X08_OUT_COL => #TEMP_X08,
            X09_OUT_COL => #TEMP_X09,
            X10_OUT_COL => #TEMP_X10,
            X11_OUT_COL => #TEMP_X11,
            X12_OUT_COL => #TEMP_X12,
            X13_OUT_COL => #TEMP_X13,
            X14_OUT_COL => #TEMP_X14,
            X15_OUT_COL => #TEMP_X15);
   "1R_TRG001" := NOT "1R_P003" AND NOT "1R_P001";   // rising edge
   "1R_P001" := NOT "1R_P003";
END_REGION

REGION Network 2
   RUNG wire#powerrail
      Contact( "1R_P001" )
      "QR_DIAG"(X00_IN_DIAG := #TEMP_X00, X01_IN_DIAG := #TEMP_X01, X02_IN_DIAG := #TEMP_X02, X03_IN_DIAG := #TEMP_X03, X04_IN_DIAG := #TEMP_X04, X05_IN_DIAG := #TEMP_X05, X06_IN_DIAG := #TEMP_X06, X07_IN_DIAG := #TEMP_X07, X08_IN_DIAG := #TEMP_X08, X09_IN_DIAG := #TEMP_X09, X10_IN_DIAG := #TEMP_X10, X11_IN_DIAG := #TEMP_X11, X12_IN_DIAG := #TEMP_X12, X13_IN_DIAG := #TEMP_X13, X14_IN_DIAG := #TEMP_X14, X15_IN_DIAG := #TEMP_X15, X00_OUT_DIAG => #X00_OUT, X01_OUT_DIAG => #X01_OUT, X02_OUT_DIAG => #X02_OUT, X03_OUT_DIAG => #X03_OUT, X04_OUT_DIAG => #X04_OUT, X05_OUT_DIAG => #X05_OUT, X06_OUT_DIAG => #X06_OUT, X07_OUT_DIAG => #X07_OUT, X08_OUT_DIAG => #X08_OUT, X09_OUT_DIAG => #X09_OUT, X10_OUT_DIAG => #X10_OUT, X11_OUT_DIAG => #X11_OUT, X12_OUT_DIAG => #X12_OUT, X13_OUT_DIAG => #X13_OUT, X14_OUT_DIAG => #X14_OUT, X15_OUT_DIAG => #X15_OUT)
   END_RUNG
   RUNG wire#powerrail
      Contact( "1R_P001" )
      R_Coil( "1R_P001" )
   END_RUNG
   // the same network as SCL:
   IF "1R_P001" THEN
       "QR_DIAG"(X00_IN_DIAG := #TEMP_X00,
                 X01_IN_DIAG := #TEMP_X01,
                 X02_IN_DIAG := #TEMP_X02,
                 X03_IN_DIAG := #TEMP_X03,
                 X04_IN_DIAG := #TEMP_X04,
                 X05_IN_DIAG := #TEMP_X05,
                 X06_IN_DIAG := #TEMP_X06,
                 X07_IN_DIAG := #TEMP_X07,
                 X08_IN_DIAG := #TEMP_X08,
                 X09_IN_DIAG := #TEMP_X09,
                 X10_IN_DIAG := #TEMP_X10,
                 X11_IN_DIAG := #TEMP_X11,
                 X12_IN_DIAG := #TEMP_X12,
                 X13_IN_DIAG := #TEMP_X13,
                 X14_IN_DIAG := #TEMP_X14,
                 X15_IN_DIAG := #TEMP_X15,
                 X00_OUT_DIAG => #X00_OUT,
                 X01_OUT_DIAG => #X01_OUT,
                 X02_OUT_DIAG => #X02_OUT,
                 X03_OUT_DIAG => #X03_OUT,
                 X04_OUT_DIAG => #X04_OUT,
                 X05_OUT_DIAG => #X05_OUT,
                 X06_OUT_DIAG => #X06_OUT,
                 X07_OUT_DIAG => #X07_OUT,
                 X08_OUT_DIAG => #X08_OUT,
                 X09_OUT_DIAG => #X09_OUT,
                 X10_OUT_DIAG => #X10_OUT,
                 X11_OUT_DIAG => #X11_OUT,
                 X12_OUT_DIAG => #X12_OUT,
                 X13_OUT_DIAG => #X13_OUT,
                 X14_OUT_DIAG => #X14_OUT,
                 X15_OUT_DIAG => #X15_OUT);
   END_IF;
   IF "1R_P001" THEN "1R_P001" := FALSE; END_IF;
END_REGION
END_FUNCTION

FUNCTION "MOVE_DATA" : Void   // FC7, LAD
{ S7_Optimized_Access := 'TRUE' }
VERSION : 0.1
   VAR_INPUT
      IN_00 : DWord;
      IN_01 : DWord;
      IN_02 : DWord;
      IN_03 : DWord;
      IN_04 : DWord;
      IN_05 : DWord;
      IN_06 : DWord;
      IN_07 : DWord;
      IN_08 : DWord;
      IN_09 : DWord;
      IN_10 : DWord;
      IN_11 : DWord;
      IN_12 : DWord;
      IN_13 : DWord;
      IN_14 : DWord;
      IN_15 : DWord;
   END_VAR
   VAR_OUTPUT
      OUT_00 : DWord;
      OUT_01 : DWord;
      OUT_02 : DWord;
      OUT_03 : DWord;
      OUT_04 : DWord;
      OUT_05 : DWord;
      OUT_06 : DWord;
      OUT_07 : DWord;
      OUT_08 : DWord;
      OUT_09 : DWord;
      OUT_10 : DWord;
      OUT_11 : DWord;
      OUT_12 : DWord;
      OUT_13 : DWord;
      OUT_14 : DWord;
      OUT_15 : DWord;
   END_VAR
BEGIN

REGION Network 1
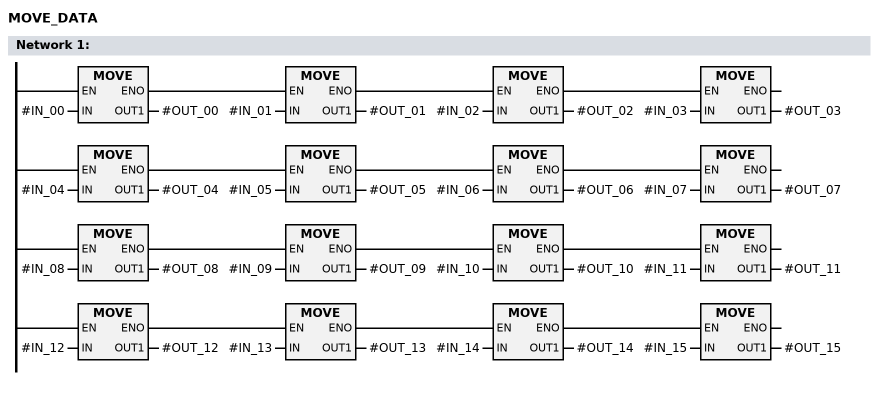
   RUNG wire#powerrail
      { S7_GenerateENO := "TRUE" } Move(in := #IN_00, out1 => #OUT_00)
      { S7_GenerateENO := "TRUE" } Move(in := #IN_01, out1 => #OUT_01)
      { S7_GenerateENO := "TRUE" } Move(in := #IN_02, out1 => #OUT_02)
      { S7_GenerateENO := "TRUE" } Move(in := #IN_03, out1 => #OUT_03)
   END_RUNG
   RUNG wire#powerrail
      { S7_GenerateENO := "TRUE" } Move(in := #IN_04, out1 => #OUT_04)
      { S7_GenerateENO := "TRUE" } Move(in := #IN_05, out1 => #OUT_05)
      { S7_GenerateENO := "TRUE" } Move(in := #IN_06, out1 => #OUT_06)
      { S7_GenerateENO := "TRUE" } Move(in := #IN_07, out1 => #OUT_07)
   END_RUNG
   RUNG wire#powerrail
      { S7_GenerateENO := "TRUE" } Move(in := #IN_08, out1 => #OUT_08)
      { S7_GenerateENO := "TRUE" } Move(in := #IN_09, out1 => #OUT_09)
      { S7_GenerateENO := "TRUE" } Move(in := #IN_10, out1 => #OUT_10)
      { S7_GenerateENO := "TRUE" } Move(in := #IN_11, out1 => #OUT_11)
   END_RUNG
   RUNG wire#powerrail
      { S7_GenerateENO := "TRUE" } Move(in := #IN_12, out1 => #OUT_12)
      { S7_GenerateENO := "TRUE" } Move(in := #IN_13, out1 => #OUT_13)
      { S7_GenerateENO := "TRUE" } Move(in := #IN_14, out1 => #OUT_14)
      { S7_GenerateENO := "TRUE" } Move(in := #IN_15, out1 => #OUT_15)
   END_RUNG
   // the same network as SCL:
   // ENO of a box is taken as its EN; it also drops when the box reports an error
   #OUT_00 := #IN_00;
   #OUT_01 := #IN_01;
   #OUT_02 := #IN_02;
   #OUT_03 := #IN_03;
   #OUT_04 := #IN_04;
   #OUT_05 := #IN_05;
   #OUT_06 := #IN_06;
   #OUT_07 := #IN_07;
   #OUT_08 := #IN_08;
   #OUT_09 := #IN_09;
   #OUT_10 := #IN_10;
   #OUT_11 := #IN_11;
   #OUT_12 := #IN_12;
   #OUT_13 := #IN_13;
   #OUT_14 := #IN_14;
   #OUT_15 := #IN_15;
END_REGION
END_FUNCTION

FUNCTION "CHACHA_EN/DECRYPT" : Void   // FC8, LAD
{ S7_Optimized_Access := 'TRUE' }
VERSION : 0.1
   VAR_INPUT
      PLAIN_IN_X00 : DWord;
      PLAIN_IN_X01 : DWord;
      PLAIN_IN_X02 : DWord;
      PLAIN_IN_X03 : DWord;
      PLAIN_IN_X04 : DWord;
      PLAIN_IN_X05 : DWord;
      PLAIN_IN_X06 : DWord;
      PLAIN_IN_X07 : DWord;
      PLAIN_IN_X08 : DWord;
      PLAIN_IN_X09 : DWord;
      PLAIN_IN_X10 : DWord;
      PLAIN_IN_X11 : DWord;
      PLAIN_IN_X12 : DWord;
      PLAIN_IN_X13 : DWord;
      PLAIN_IN_X14 : DWord;
      PLAIN_IN_X15 : DWord;
      KSTRM_IN_X00 : DWord;
      KSTRM_IN_X01 : DWord;
      KSTRM_IN_X02 : DWord;
      KSTRM_IN_X03 : DWord;
      KSTRM_IN_X04 : DWord;
      KSTRM_IN_X05 : DWord;
      KSTRM_IN_X06 : DWord;
      KSTRM_IN_X07 : DWord;
      KSTRM_IN_X08 : DWord;
      KSTRM_IN_X09 : DWord;
      KSTRM_IN_X10 : DWord;
      KSTRM_IN_X11 : DWord;
      KSTRM_IN_X12 : DWord;
      KSTRM_IN_X13 : DWord;
      KSTRM_IN_X14 : DWord;
      KSTRM_IN_X15 : DWord;
   END_VAR
   VAR_OUTPUT
      CIPHERTXT_OUT_X00 : DWord;
      CIPHERTXT_OUT_X01 : DWord;
      CIPHERTXT_OUT_X02 : DWord;
      CIPHERTXT_OUT_X03 : DWord;
      CIPHERTXT_OUT_X04 : DWord;
      CIPHERTXT_OUT_X05 : DWord;
      CIPHERTXT_OUT_X06 : DWord;
      CIPHERTXT_OUT_X07 : DWord;
      CIPHERTXT_OUT_X08 : DWord;
      CIPHERTXT_OUT_X09 : DWord;
      CIPHERTXT_OUT_X10 : DWord;
      CIPHERTXT_OUT_X11 : DWord;
      CIPHERTXT_OUT_X12 : DWord;
      CIPHERTXT_OUT_X13 : DWord;
      CIPHERTXT_OUT_X14 : DWord;
      CIPHERTXT_OUT_X15 : DWord;
   END_VAR
BEGIN

REGION Network 1
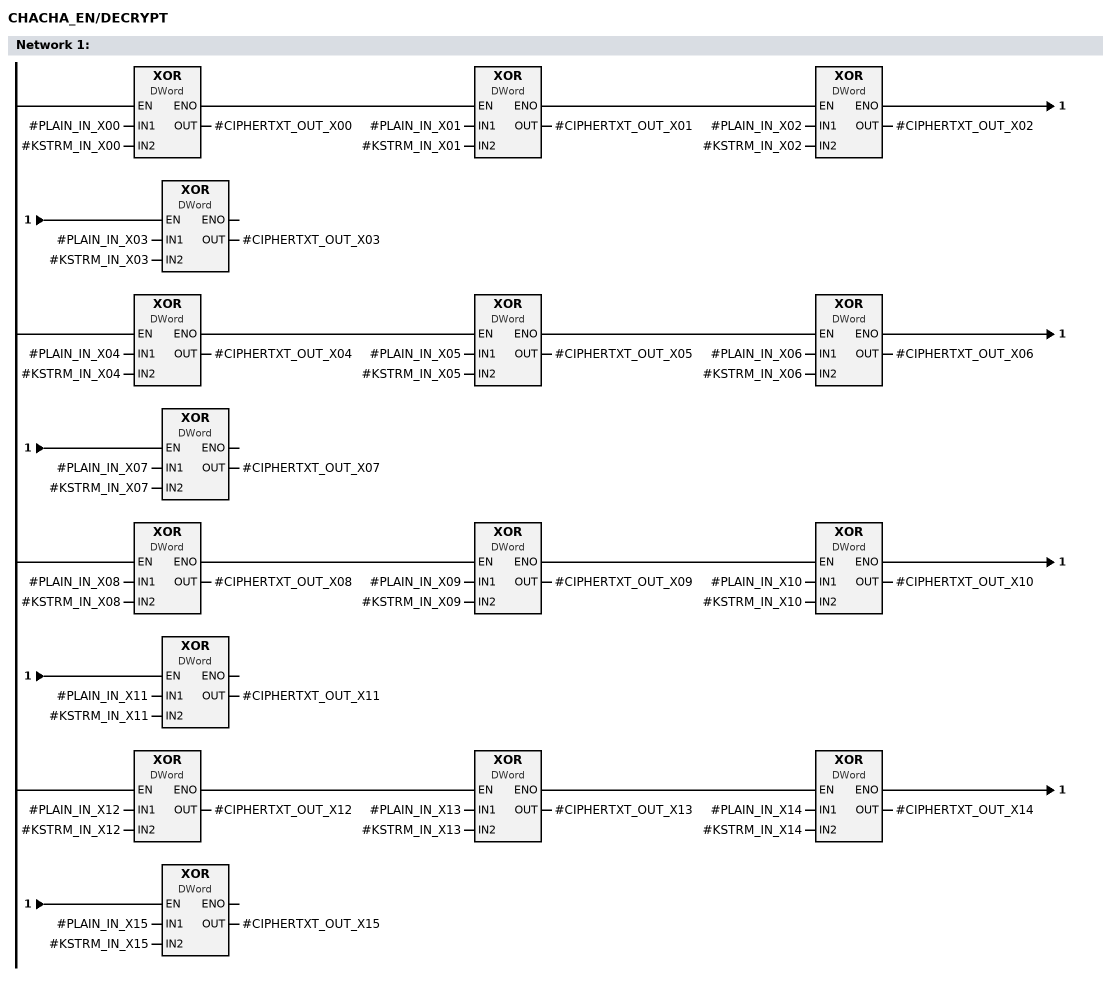
   #CIPHERTXT_OUT_X00 := #PLAIN_IN_X00 XOR #KSTRM_IN_X00;
   #CIPHERTXT_OUT_X01 := #PLAIN_IN_X01 XOR #KSTRM_IN_X01;
   #CIPHERTXT_OUT_X02 := #PLAIN_IN_X02 XOR #KSTRM_IN_X02;
   #CIPHERTXT_OUT_X03 := #PLAIN_IN_X03 XOR #KSTRM_IN_X03;
   #CIPHERTXT_OUT_X04 := #PLAIN_IN_X04 XOR #KSTRM_IN_X04;
   #CIPHERTXT_OUT_X05 := #PLAIN_IN_X05 XOR #KSTRM_IN_X05;
   #CIPHERTXT_OUT_X06 := #PLAIN_IN_X06 XOR #KSTRM_IN_X06;
   #CIPHERTXT_OUT_X07 := #PLAIN_IN_X07 XOR #KSTRM_IN_X07;
   #CIPHERTXT_OUT_X08 := #PLAIN_IN_X08 XOR #KSTRM_IN_X08;
   #CIPHERTXT_OUT_X09 := #PLAIN_IN_X09 XOR #KSTRM_IN_X09;
   #CIPHERTXT_OUT_X10 := #PLAIN_IN_X10 XOR #KSTRM_IN_X10;
   #CIPHERTXT_OUT_X11 := #PLAIN_IN_X11 XOR #KSTRM_IN_X11;
   #CIPHERTXT_OUT_X12 := #PLAIN_IN_X12 XOR #KSTRM_IN_X12;
   #CIPHERTXT_OUT_X13 := #PLAIN_IN_X13 XOR #KSTRM_IN_X13;
   #CIPHERTXT_OUT_X14 := #PLAIN_IN_X14 XOR #KSTRM_IN_X14;
   #CIPHERTXT_OUT_X15 := #PLAIN_IN_X15 XOR #KSTRM_IN_X15;
END_REGION
END_FUNCTION

FUNCTION "ADD_DWORD" : Void   // FC9, LAD
{ S7_Optimized_Access := 'TRUE' }
VERSION : 0.1
   VAR_INPUT
      IN_A00 : DWord;
      IN_A01 : DWord;
      IN_A02 : DWord;
      IN_A03 : DWord;
      IN_A04 : DWord;
      IN_A05 : DWord;
      IN_A06 : DWord;
      IN_A07 : DWord;
      IN_A08 : DWord;
      IN_A09 : DWord;
      IN_A10 : DWord;
      IN_A11 : DWord;
      IN_A12 : DWord;
      IN_A13 : DWord;
      IN_A14 : DWord;
      IN_A15 : DWord;
      IN_B00 : DWord;
      IN_B01 : DWord;
      IN_B02 : DWord;
      IN_B03 : DWord;
      IN_B04 : DWord;
      IN_B05 : DWord;
      IN_B06 : DWord;
      IN_B07 : DWord;
      IN_B08 : DWord;
      IN_B09 : DWord;
      IN_B10 : DWord;
      IN_B11 : DWord;
      IN_B12 : DWord;
      IN_B13 : DWord;
      IN_B14 : DWord;
      IN_B15 : DWord;
   END_VAR
   VAR_OUTPUT
      OUT_00 : DWord;
      OUT_01 : DWord;
      OUT_02 : DWord;
      OUT_03 : DWord;
      OUT_04 : DWord;
      OUT_05 : DWord;
      OUT_06 : DWord;
      OUT_07 : DWord;
      OUT_08 : DWord;
      OUT_09 : DWord;
      OUT_10 : DWord;
      OUT_11 : DWord;
      OUT_12 : DWord;
      OUT_13 : DWord;
      OUT_14 : DWord;
      OUT_15 : DWord;
   END_VAR
   VAR_TEMP
      A0 : UDInt;
      A1 : UDInt;
      A2 : UDInt;
      A3 : UDInt;
      A4 : UDInt;
      A5 : UDInt;
      A6 : UDInt;
      A7 : UDInt;
      A8 : UDInt;
      A9 : UDInt;
      A10 : UDInt;
      A11 : UDInt;
      A12 : UDInt;
      A13 : UDInt;
      A14 : UDInt;
      A15 : UDInt;
      B0 : UDInt;
      B1 : UDInt;
      B2 : UDInt;
      B3 : UDInt;
      B4 : UDInt;
      B5 : UDInt;
      B6 : UDInt;
      B7 : UDInt;
      B8 : UDInt;
      B9 : UDInt;
      B10 : UDInt;
      B11 : UDInt;
      B12 : UDInt;
      B13 : UDInt;
      B14 : UDInt;
      B15 : UDInt;
      R0 : UDInt;
      R1 : UDInt;
      R2 : UDInt;
      R3 : UDInt;
      R4 : UDInt;
      R5 : UDInt;
      R6 : UDInt;
      R7 : UDInt;
      R8 : UDInt;
      R9 : UDInt;
      R10 : UDInt;
      R11 : UDInt;
      R12 : UDInt;
      R13 : UDInt;
      R14 : UDInt;
      R15 : UDInt;
   END_VAR
   VAR_TEMP   // added for the SCL form of the ladder/FBD networks
      _w1 : Bool;
      _w2 : Bool;
   END_VAR
BEGIN

REGION Network 1
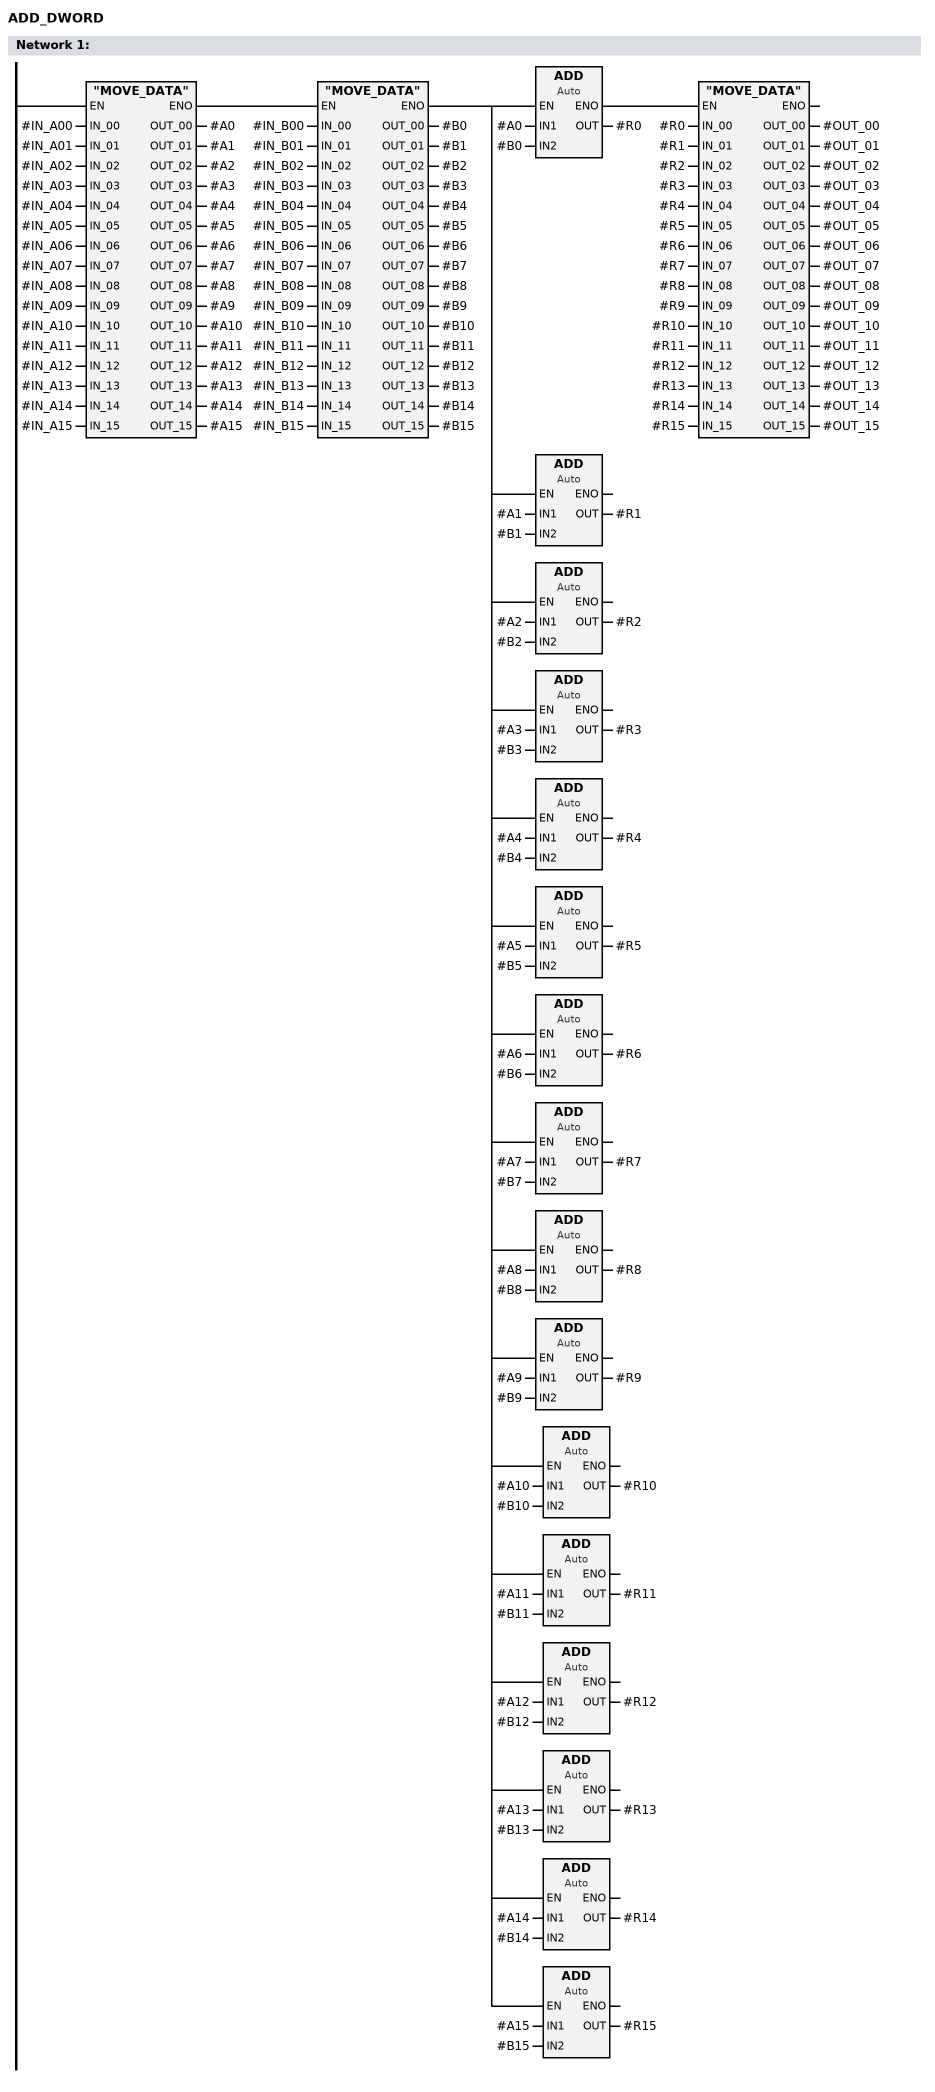
   RUNG wire#powerrail
      "MOVE_DATA"(IN_00 := #IN_A00, IN_01 := #IN_A01, IN_02 := #IN_A02, IN_03 := #IN_A03, IN_04 := #IN_A04, IN_05 := #IN_A05, IN_06 := #IN_A06, IN_07 := #IN_A07, IN_08 := #IN_A08, IN_09 := #IN_A09, IN_10 := #IN_A10, IN_11 := #IN_A11, IN_12 := #IN_A12, IN_13 := #IN_A13, IN_14 := #IN_A14, IN_15 := #IN_A15, OUT_00 => #A0, OUT_01 => #A1, OUT_02 => #A2, OUT_03 => #A3, OUT_04 => #A4, OUT_05 => #A5, OUT_06 => #A6, OUT_07 => #A7, OUT_08 => #A8, OUT_09 => #A9, OUT_10 => #A10, OUT_11 => #A11, OUT_12 => #A12, OUT_13 => #A13, OUT_14 => #A14, OUT_15 => #A15)
      "MOVE_DATA"(IN_00 := #IN_B00, IN_01 := #IN_B01, IN_02 := #IN_B02, IN_03 := #IN_B03, IN_04 := #IN_B04, IN_05 := #IN_B05, IN_06 := #IN_B06, IN_07 := #IN_B07, IN_08 := #IN_B08, IN_09 := #IN_B09, IN_10 := #IN_B10, IN_11 := #IN_B11, IN_12 := #IN_B12, IN_13 := #IN_B13, IN_14 := #IN_B14, IN_15 := #IN_B15, OUT_00 => #B0, OUT_01 => #B1, OUT_02 => #B2, OUT_03 => #B3, OUT_04 => #B4, OUT_05 => #B5, OUT_06 => #B6, OUT_07 => #B7, OUT_08 => #B8, OUT_09 => #B9, OUT_10 => #B10, OUT_11 => #B11, OUT_12 => #B12, OUT_13 => #B13, OUT_14 => #B14, OUT_15 => #B15)
      wire#w1
      { S7_GenerateENO := "TRUE" } Add(in1 := #A0, in2 := #B0, out => #R0)
      "MOVE_DATA"(IN_00 := #R0, IN_01 := #R1, IN_02 := #R2, IN_03 := #R3, IN_04 := #R4, IN_05 := #R5, IN_06 := #R6, IN_07 := #R7, IN_08 := #R8, IN_09 := #R9, IN_10 := #R10, IN_11 := #R11, IN_12 := #R12, IN_13 := #R13, IN_14 := #R14, IN_15 := #R15, OUT_00 => #OUT_00, OUT_01 => #OUT_01, OUT_02 => #OUT_02, OUT_03 => #OUT_03, OUT_04 => #OUT_04, OUT_05 => #OUT_05, OUT_06 => #OUT_06, OUT_07 => #OUT_07, OUT_08 => #OUT_08, OUT_09 => #OUT_09, OUT_10 => #OUT_10, OUT_11 => #OUT_11, OUT_12 => #OUT_12, OUT_13 => #OUT_13, OUT_14 => #OUT_14, OUT_15 => #OUT_15)
   END_RUNG
   RUNG wire#w1
      { S7_GenerateENO := "TRUE" } Add(in1 := #A1, in2 := #B1, out => #R1)
   END_RUNG
   RUNG wire#w1
      { S7_GenerateENO := "TRUE" } Add(in1 := #A2, in2 := #B2, out => #R2)
   END_RUNG
   RUNG wire#w1
      { S7_GenerateENO := "TRUE" } Add(in1 := #A3, in2 := #B3, out => #R3)
   END_RUNG
   RUNG wire#w1
      { S7_GenerateENO := "TRUE" } Add(in1 := #A4, in2 := #B4, out => #R4)
   END_RUNG
   RUNG wire#w1
      { S7_GenerateENO := "TRUE" } Add(in1 := #A5, in2 := #B5, out => #R5)
   END_RUNG
   RUNG wire#w1
      { S7_GenerateENO := "TRUE" } Add(in1 := #A6, in2 := #B6, out => #R6)
   END_RUNG
   RUNG wire#w1
      { S7_GenerateENO := "TRUE" } Add(in1 := #A7, in2 := #B7, out => #R7)
   END_RUNG
   RUNG wire#w1
      { S7_GenerateENO := "TRUE" } Add(in1 := #A8, in2 := #B8, out => #R8)
   END_RUNG
   RUNG wire#w1
      { S7_GenerateENO := "TRUE" } Add(in1 := #A9, in2 := #B9, out => #R9)
   END_RUNG
   RUNG wire#w1
      { S7_GenerateENO := "TRUE" } Add(in1 := #A10, in2 := #B10, out => #R10)
   END_RUNG
   RUNG wire#w1
      { S7_GenerateENO := "TRUE" } Add(in1 := #A11, in2 := #B11, out => #R11)
   END_RUNG
   RUNG wire#w1
      { S7_GenerateENO := "TRUE" } Add(in1 := #A12, in2 := #B12, out => #R12)
   END_RUNG
   RUNG wire#w1
      { S7_GenerateENO := "TRUE" } Add(in1 := #A13, in2 := #B13, out => #R13)
   END_RUNG
   RUNG wire#w1
      { S7_GenerateENO := "TRUE" } Add(in1 := #A14, in2 := #B14, out => #R14)
   END_RUNG
   RUNG wire#w1
      { S7_GenerateENO := "TRUE" } Add(in1 := #A15, in2 := #B15, out => #R15)
   END_RUNG
   // the same network as SCL:
   // ENO of a box is taken as its EN; it also drops when the box reports an error
   "MOVE_DATA"(IN_00 := #IN_A00,
               IN_01 := #IN_A01,
               IN_02 := #IN_A02,
               IN_03 := #IN_A03,
               IN_04 := #IN_A04,
               IN_05 := #IN_A05,
               IN_06 := #IN_A06,
               IN_07 := #IN_A07,
               IN_08 := #IN_A08,
               IN_09 := #IN_A09,
               IN_10 := #IN_A10,
               IN_11 := #IN_A11,
               IN_12 := #IN_A12,
               IN_13 := #IN_A13,
               IN_14 := #IN_A14,
               IN_15 := #IN_A15,
               OUT_00 => #A0,
               OUT_01 => #A1,
               OUT_02 => #A2,
               OUT_03 => #A3,
               OUT_04 => #A4,
               OUT_05 => #A5,
               OUT_06 => #A6,
               OUT_07 => #A7,
               OUT_08 => #A8,
               OUT_09 => #A9,
               OUT_10 => #A10,
               OUT_11 => #A11,
               OUT_12 => #A12,
               OUT_13 => #A13,
               OUT_14 => #A14,
               OUT_15 => #A15,
               ENO => #_w1);
   "MOVE_DATA"(EN := #_w1,
               IN_00 := #IN_B00,
               IN_01 := #IN_B01,
               IN_02 := #IN_B02,
               IN_03 := #IN_B03,
               IN_04 := #IN_B04,
               IN_05 := #IN_B05,
               IN_06 := #IN_B06,
               IN_07 := #IN_B07,
               IN_08 := #IN_B08,
               IN_09 := #IN_B09,
               IN_10 := #IN_B10,
               IN_11 := #IN_B11,
               IN_12 := #IN_B12,
               IN_13 := #IN_B13,
               IN_14 := #IN_B14,
               IN_15 := #IN_B15,
               OUT_00 => #B0,
               OUT_01 => #B1,
               OUT_02 => #B2,
               OUT_03 => #B3,
               OUT_04 => #B4,
               OUT_05 => #B5,
               OUT_06 => #B6,
               OUT_07 => #B7,
               OUT_08 => #B8,
               OUT_09 => #B9,
               OUT_10 => #B10,
               OUT_11 => #B11,
               OUT_12 => #B12,
               OUT_13 => #B13,
               OUT_14 => #B14,
               OUT_15 => #B15,
               ENO => #_w2);
   IF #_w2 THEN
       #R0 := #A0 + #B0;
       "MOVE_DATA"(IN_00 := #R0,
                   IN_01 := #R1,
                   IN_02 := #R2,
                   IN_03 := #R3,
                   IN_04 := #R4,
                   IN_05 := #R5,
                   IN_06 := #R6,
                   IN_07 := #R7,
                   IN_08 := #R8,
                   IN_09 := #R9,
                   IN_10 := #R10,
                   IN_11 := #R11,
                   IN_12 := #R12,
                   IN_13 := #R13,
                   IN_14 := #R14,
                   IN_15 := #R15,
                   OUT_00 => #OUT_00,
                   OUT_01 => #OUT_01,
                   OUT_02 => #OUT_02,
                   OUT_03 => #OUT_03,
                   OUT_04 => #OUT_04,
                   OUT_05 => #OUT_05,
                   OUT_06 => #OUT_06,
                   OUT_07 => #OUT_07,
                   OUT_08 => #OUT_08,
                   OUT_09 => #OUT_09,
                   OUT_10 => #OUT_10,
                   OUT_11 => #OUT_11,
                   OUT_12 => #OUT_12,
                   OUT_13 => #OUT_13,
                   OUT_14 => #OUT_14,
                   OUT_15 => #OUT_15);
       #R1 := #A1 + #B1;
       #R2 := #A2 + #B2;
       #R3 := #A3 + #B3;
       #R4 := #A4 + #B4;
       #R5 := #A5 + #B5;
       #R6 := #A6 + #B6;
       #R7 := #A7 + #B7;
       #R8 := #A8 + #B8;
       #R9 := #A9 + #B9;
       #R10 := #A10 + #B10;
       #R11 := #A11 + #B11;
       #R12 := #A12 + #B12;
       #R13 := #A13 + #B13;
       #R14 := #A14 + #B14;
       #R15 := #A15 + #B15;
   END_IF;
END_REGION
END_FUNCTION

ORGANIZATION_BLOCK "Main"   // OB1, LAD, ProgramCycle
TITLE = "Main Program Sweep (Cycle)"
{ S7_Optimized_Access := 'TRUE' }
VERSION : 0.1
   VAR_TEMP   // added for the SCL form of the ladder/FBD networks
      _w1 : Bool;
      _w2 : Bool;
      _w3 : Bool;
      _w4 : Bool;
   END_VAR
BEGIN

REGION Network 1: TESTE CHACHA 20 ROUNDS - RUNTIME START
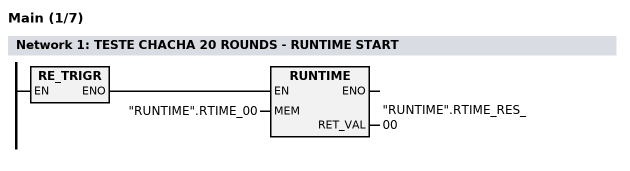
   // no SCL statement known for Runtime: written as a call
   // ENO of a box is taken as its EN; it also drops when the box reports an error
   RE_TRIGR();
   "RUNTIME".RTIME_RES_00 := Runtime(mem := "RUNTIME".RTIME_00);
END_REGION

